LIN {X 0,Y 156.804,Z 513.248,A -85,B 0,C 180,E1 -23850.002,E2 -23850.002} C_VEL
LIN {X 0,Y 156.552,Z 512.223,A -85,B 0,C 180,E1 -23852.575,E2 -23852.575} C_VEL
LIN {X 0,Y 156.139,Z 510.706,A -85,B 0,C 180,E1 -23855.167,E2 -23855.167} C_VEL
LIN {X 0,Y 155.903,Z 507.578,A -85,B 0,C 180,E1 -23859.08,E2 -23859.08} C_VEL
LIN {X 0,Y 156.234,Z 503.359,A -85,B 0,C 180,E1 -23863,E2 -23863} C_VEL
LIN {X 0,Y 157.456,Z 496.901,A -85,B 0,C 180,E1 -23867.537,E2 -23867.537} C_VEL
LIN {X 0,Y 159.345,Z 489.978,A -85,B 0,C 180,E1 -23871.306,E2 -23871.306} C_VEL
LIN {X 0,Y 161.489,Z 483.128,A -85,B 0,C 180,E1 -23874.286,E2 -23874.286} C_VEL
LIN {X 0,Y 162.926,Z 474.015,A -85,B 0,C 180,E1 -23877.629,E2 -23877.629} C_VEL
LIN {X 0,Y 164.364,Z 464.341,A -85,B 0,C 180,E1 -23880.517,E2 -23880.517} C_VEL
LIN {X 0,Y 165.396,Z 453.516,A -85,B 0,C 180,E1 -23883.204,E2 -23883.204} C_VEL
LIN {X 0,Y 165.775,Z 447.367,A -85,B 0,C 180,E1 -23884.528,E2 -23884.528} C_VEL
LIN {X 0,Y 165.255,Z 442.446,A -85,B 0,C 180,E1 -23885.654,E2 -23885.654} C_VEL
LIN {X 0,Y 162.511,Z 434.79,A -85,B 0,C 180,E1 -23887.665,E2 -23887.665} C_VEL
LIN {X 0,Y 159.533,Z 426.921,A -85,B 0,C 180,E1 -23889.587,E2 -23889.587} C_VEL
LIN {X 0,Y 158.608,Z 421.658,A -85,B 0,C 180,E1 -23890.529,E2 -23890.529} C_VEL
LIN {X 0,Y 157.114,Z 411.985,A -85,B 0,C 180,E1 -23892.069,E2 -23892.069} C_VEL
LIN {X 0,Y 154.902,Z 406.011,A -85,B 0,C 180,E1 -23893.256,E2 -23893.256} C_VEL
LIN {X 0,Y 153.361,Z 402.44,A -85,B 0,C 180,E1 -23893.995,E2 -23893.995} C_VEL
LIN {X 0,Y 153.171,Z 401.481,A -85,B 0,C 180,E1 -23894.172,E2 -23894.172} C_VEL
LIN {X 0,Y 152.154,Z 396.368,A -85,B 0,C 180,E1 -23899.71,E2 -23899.71} C_VEL
LIN {X 0,Y 151.356,Z 392.231,A -85,B 0,C 180,E1 -23904.52,E2 -23904.52} C_VEL
LIN {X 0,Y 150.667,Z 388.552,A -85,B 0,C 180,E1 -23909.13,E2 -23909.13} C_VEL
LIN {X 0,Y 150.262,Z 386.768,A -85,B 0,C 180,E1 -23911.735,E2 -23911.735} C_VEL
LIN {X 0,Y 150.274,Z 386.771,A -85,B 0,C 180,E1 -23918.029,E2 -23918.029} C_VEL
LIN {X 0,Y 150.378,Z 386.759,A -85,B 0,C 180,E1 -23920.905,E2 -23920.905} C_VEL
LIN {X 0,Y 150.473,Z 386.744,A -85,B 0,C 180,E1 -23926.496,E2 -23926.496} C_VEL
LIN {X 0,Y 150.695,Z 386.714,A -85,B 0,C 180,E1 -23929.249,E2 -23929.249} C_VEL
LIN {X 0,Y 150.769,Z 386.706,A -85,B 0,C 180,E1 -23931.962,E2 -23931.962} C_VEL
LIN {X 0,Y 151.225,Z 386.636,A -85,B 0,C 180,E1 -23940.001,E2 -23940.001} C_VEL
LIN {X 0,Y 150.767,Z 386.689,A -85,B 0,C 180,E1 -23948.04,E2 -23948.04} C_VEL
LIN {X 0,Y 150.64,Z 386.72,A -85,B 0,C 180,E1 -23951.545,E2 -23951.545} C_VEL
LIN {X 0,Y 150.374,Z 386.739,A -85,B 0,C 180,E1 -23956.286,E2 -23956.286} C_VEL
LIN {X 0,Y 150.357,Z 386.752,A -85,B 0,C 180,E1 -23960.793,E2 -23960.793} C_VEL
LIN {X 0,Y 150.251,Z 386.77,A -85,B 0,C 180,E1 -23967.282,E2 -23967.282} C_VEL
LIN {X 0,Y 150.225,Z 386.771,A -85,B 0,C 180,E1 -23972.634,E2 -23972.634} C_VEL
LIN {X 0,Y 150.217,Z 386.772,A -85,B 0,C 180,E1 -23977.461,E2 -23977.461} C_VEL
LIN {X 0,Y 150.16,Z 386.776,A -85,B 0,C 180,E1 -23981.506,E2 -23981.506} C_VEL
LIN {X 0,Y 150.131,Z 386.78,A -85,B 0,C 180,E1 -23985.395,E2 -23985.395} C_VEL
LIN {X 0,Y 150.156,Z 386.778,A -85,B 0,C 180,E1 -23989.058,E2 -23989.058} C_VEL
LIN {X 0,Y 150.282,Z 386.884,A -85,B 0,C 180,E1 -23994.46,E2 -23994.46} C_VEL
LIN {X 0,Y 151.235,Z 389.587,A -85,B 0,C 180,E1 -23995.172,E2 -23995.172} C_VEL
LIN {X 0,Y 152.671,Z 391.781,A -85,B 0,C 180,E1 -23995.957,E2 -23995.957} C_VEL
LIN {X 0,Y 157.325,Z 400.956,A -85,B 0,C 180,E1 -23998.953,E2 -23998.953} C_VEL
LIN {X 0,Y 161.282,Z 410.794,A -85,B 0,C 180,E1 -24002.092,E2 -24002.092} C_VEL
LIN {X 0,Y 164.08,Z 420.392,A -85,B 0,C 180,E1 -24005.202,E2 -24005.202} C_VEL
LIN {X 0,Y 165.343,Z 425.976,A -85,B 0,C 180,E1 -24007.113,E2 -24007.113} C_VEL
LIN {X 0,Y 162.841,Z 435.568,A -85,B 0,C 180,E1 -24009.8,E2 -24009.8} C_VEL
LIN {X 0,Y 160.103,Z 444.185,A -85,B 0,C 180,E1 -24012.762,E2 -24012.762} C_VEL
LIN {X 0,Y 157.588,Z 451.322,A -85,B 0,C 180,E1 -24015.799,E2 -24015.799} C_VEL
LIN {X 0,Y 155.089,Z 458.345,A -85,B 0,C 180,E1 -24019.555,E2 -24019.555} C_VEL
LIN {X 0,Y 153.157,Z 463.944,A -85,B 0,C 180,E1 -24023.411,E2 -24023.411} C_VEL
LIN {X 0,Y 151.613,Z 468.389,A -85,B 0,C 180,E1 -24027.341,E2 -24027.341} C_VEL
LIN {X 0,Y 150.875,Z 470.747,A -85,B 0,C 180,E1 -24029.998,E2 -24029.998} C_VEL
LIN {X 0,Y 150.369,Z 472.687,A -85,B 0,C 180,E1 -24032.677,E2 -24032.677} C_VEL
LIN {X 0,Y 150.284,Z 474.186,A -85,B 0,C 180,E1 -24035.365,E2 -24035.365} C_VEL
LIN {X 0,Y 150.347,Z 475.258,A -85,B 0,C 180,E1 -24038.06,E2 -24038.06} C_VEL
LIN {X 0,Y 151.03,Z 476.287,A -85,B 0,C 180,E1 -24043.452,E2 -24043.452} C_VEL
LIN {X 0,Y 151.721,Z 476.222,A -85,B 0,C 180,E1 -24046.135,E2 -24046.135} C_VEL
LIN {X 0,Y 153.88,Z 474.85,A -85,B 0,C 180,E1 -24051.429,E2 -24051.429} C_VEL
LIN {X 0,Y 155.422,Z 473.57,A -85,B 0,C 180,E1 -24054.012,E2 -24054.012} C_VEL
LIN {X 0,Y 158.105,Z 470.825,A -85,B 0,C 180,E1 -24057.821,E2 -24057.821} C_VEL
LIN {X 0,Y 161.348,Z 467.038,A -85,B 0,C 180,E1 -24061.511,E2 -24061.511} C_VEL
LIN {X 0,Y 165.108,Z 462.098,A -85,B 0,C 180,E1 -24065.072,E2 -24065.072} C_VEL
LIN {X 0,Y 169.45,Z 455.8,A -85,B 0,C 180,E1 -24068.47,E2 -24068.47} C_VEL
LIN {X 0,Y 174.228,Z 447.87,A -85,B 0,C 180,E1 -24071.724,E2 -24071.724} C_VEL
LIN {X 0,Y 175.852,Z 444.813,A -85,B 0,C 180,E1 -24072.795,E2 -24072.795} C_VEL
LIN {X 0,Y 175.242,Z 438.143,A -85,B 0,C 180,E1 -24076.208,E2 -24076.208} C_VEL
LIN {X 0,Y 173.539,Z 430.026,A -85,B 0,C 180,E1 -24080.303,E2 -24080.303} C_VEL
LIN {X 0,Y 171.262,Z 422.341,A -85,B 0,C 180,E1 -24084.212,E2 -24084.212} C_VEL
LIN {X 0,Y 168.083,Z 414.609,A -85,B 0,C 180,E1 -24088.488,E2 -24088.488} C_VEL
LIN {X 0,Y 164.176,Z 406.916,A -85,B 0,C 180,E1 -24093.289,E2 -24093.289} C_VEL
LIN {X 0,Y 161.151,Z 402.126,A -85,B 0,C 180,E1 -24096.889,E2 -24096.889} C_VEL
LIN {X 0,Y 159.253,Z 399.15,A -85,B 0,C 180,E1 -24099.325,E2 -24099.325} C_VEL
LIN {X 0,Y 158.101,Z 397.442,A -85,B 0,C 180,E1 -24100.862,E2 -24100.862} C_VEL
LIN {X 0,Y 156.068,Z 395.021,A -85,B 0,C 180,E1 -24103.653,E2 -24103.653} C_VEL
LIN {X 0,Y 155.062,Z 392.527,A -85,B 0,C 180,E1 -24105.564,E2 -24105.564} C_VEL
LIN {X 0,Y 152.252,Z 390.308,A -85,B 0,C 180,E1 -24110.367,E2 -24110.367} C_VEL
LIN {X 0,Y 150.758,Z 387.15,A -85,B 0,C 180,E1 -24114.817,E2 -24114.817} C_VEL
LIN {X 0,Y 150.713,Z 386.693,A -85,B 0,C 180,E1 -24115.319,E2 -24115.319} C_VEL
LIN {X 0,Y 151.218,Z 386.63,A -85,B 0,C 180,E1 -24119.999,E2 -24119.999} C_VEL
LIN {X 0,Y 150.955,Z 386.816,A -85,B 0,C 180,E1 -24122.668,E2 -24122.668} C_VEL
LIN {X 0,Y 151.141,Z 388.563,A -85,B 0,C 180,E1 -24128.018,E2 -24128.018} C_VEL
LIN {X 0,Y 151.34,Z 389.576,A -85,B 0,C 180,E1 -24130.705,E2 -24130.705} C_VEL
LIN {X 0,Y 151.465,Z 391.249,A -85,B 0,C 180,E1 -24134.099,E2 -24134.099} C_VEL
LIN {X 0,Y 154.139,Z 397.245,A -85,B 0,C 180,E1 -24139.649,E2 -24139.649} C_VEL
LIN {X 0,Y 156.992,Z 401.179,A -85,B 0,C 180,E1 -24143.54,E2 -24143.54} C_VEL
LIN {X 0,Y 158.698,Z 405.379,A -85,B 0,C 180,E1 -24145.932,E2 -24145.932} C_VEL
LIN {X 0,Y 161.296,Z 409.223,A -85,B 0,C 180,E1 -24148.69,E2 -24148.69} C_VEL
LIN {X 0,Y 163.364,Z 414.032,A -85,B 0,C 180,E1 -24151.08,E2 -24151.08} C_VEL
LIN {X 0,Y 164.608,Z 416.098,A -85,B 0,C 180,E1 -24152.255,E2 -24152.255} C_VEL
LIN {X 0,Y 165.981,Z 419.751,A -85,B 0,C 180,E1 -24153.832,E2 -24153.832} C_VEL
LIN {X 0,Y 167.386,Z 422.972,A -85,B 0,C 180,E1 -24155.262,E2 -24155.262} C_VEL
LIN {X 0,Y 169.635,Z 429.16,A -85,B 0,C 180,E1 -24157.744,E2 -24157.744} C_VEL
LIN {X 0,Y 172.193,Z 437.216,A -85,B 0,C 180,E1 -24160.77,E2 -24160.77} C_VEL
LIN {X 0,Y 172.884,Z 439.902,A -85,B 0,C 180,E1 -24161.71,E2 -24161.71} C_VEL
LIN {X 0,Y 172.455,Z 450.46,A -85,B 0,C 180,E1 -24164.471,E2 -24164.471} C_VEL
LIN {X 0,Y 171.024,Z 461.95,A -85,B 0,C 180,E1 -24167.704,E2 -24167.704} C_VEL
LIN {X 0,Y 169.027,Z 471.309,A -85,B 0,C 180,E1 -24170.65,E2 -24170.65} C_VEL
LIN {X 0,Y 166.508,Z 479.96,A -85,B 0,C 180,E1 -24173.78,E2 -24173.78} C_VEL
LIN {X 0,Y 163.75,Z 487.195,A -85,B 0,C 180,E1 -24176.826,E2 -24176.826} C_VEL
LIN {X 0,Y 160.277,Z 493.196,A -85,B 0,C 180,E1 -24179.72,E2 -24179.72} C_VEL
LIN {X 0,Y 156.417,Z 499.094,A -85,B 0,C 180,E1 -24183.303,E2 -24183.303} C_VEL
LIN {X 0,Y 153.318,Z 503.813,A -85,B 0,C 180,E1 -24187.07,E2 -24187.07} C_VEL
LIN {X 0,Y 151.006,Z 507.478,A -85,B 0,C 180,E1 -24190.989,E2 -24190.989} C_VEL
LIN {X 0,Y 149.135,Z 510.845,A -85,B 0,C 180,E1 -24196.374,E2 -24196.374} C_VEL
LIN {X 0,Y 148.732,Z 512.676,A -85,B 0,C 180,E1 -24201.852,E2 -24201.852} C_VEL
LIN {X 0,Y 148.981,Z 512.974,A -85,B 0,C 180,E1 -24204.588,E2 -24204.588} C_VEL
LIN {X 0,Y 149.486,Z 512.875,A -85,B 0,C 180,E1 -24207.307,E2 -24207.307} C_VEL
LIN {X 0,Y 149.755,Z 512.326,A -85,B 0,C 180,E1 -24210.002,E2 -24210.002} C_VEL
LIN {X 0,Y 149.455,Z 511.273,A -85,B 0,C 180,E1 -24212.697,E2 -24212.697} C_VEL
LIN {X 0,Y 148.909,Z 508.114,A -85,B 0,C 180,E1 -24217.64,E2 -24217.64} C_VEL
LIN {X 0,Y 149.055,Z 503.801,A -85,B 0,C 180,E1 -24222.252,E2 -24222.252} C_VEL
LIN {X 0,Y 149.915,Z 498.753,A -85,B 0,C 180,E1 -24226.339,E2 -24226.339} C_VEL
LIN {X 0,Y 151.489,Z 492.41,A -85,B 0,C 180,E1 -24230.364,E2 -24230.364} C_VEL
LIN {X 0,Y 154.137,Z 484.605,A -85,B 0,C 180,E1 -24234.23,E2 -24234.23} C_VEL
LIN {X 0,Y 155.227,Z 479.875,A -85,B 0,C 180,E1 -24236.198,E2 -24236.198} C_VEL
LIN {X 0,Y 156.894,Z 469.535,A -85,B 0,C 180,E1 -24239.892,E2 -24239.892} C_VEL
LIN {X 0,Y 158.385,Z 459.298,A -85,B 0,C 180,E1 -24242.853,E2 -24242.853} C_VEL
LIN {X 0,Y 159.327,Z 448.053,A -85,B 0,C 180,E1 -24245.558,E2 -24245.558} C_VEL
LIN {X 0,Y 159.587,Z 437.505,A -85,B 0,C 180,E1 -24247.724,E2 -24247.724} C_VEL
LIN {X 0,Y 158.895,Z 424.497,A -85,B 0,C 180,E1 -24250.053,E2 -24250.053} C_VEL
LIN {X 0,Y 158.608,Z 421.658,A -85,B 0,C 180,E1 -24250.529,E2 -24250.529} C_VEL
LIN {X 0,Y 157.656,Z 418.369,A -85,B 0,C 180,E1 -24251.197,E2 -24251.197} C_VEL
LIN {X 0,Y 155.771,Z 415.711,A -85,B 0,C 180,E1 -24252.036,E2 -24252.036} C_VEL
LIN {X 0,Y 150.382,Z 410.253,A -85,B 0,C 180,E1 -24254.212,E2 -24254.212} C_VEL
LIN {X 0,Y 148.643,Z 407.257,A -85,B 0,C 180,E1 -24255.055,E2 -24255.055} C_VEL
LIN {X 0,Y 147.84,Z 405.365,A -85,B 0,C 180,E1 -24255.501,E2 -24255.501} C_VEL
LIN {X 0,Y 146.067,Z 401.9,A -85,B 0,C 180,E1 -24256.411,E2 -24256.411} C_VEL
LIN {X 0,Y 145.648,Z 400.322,A -85,B 0,C 180,E1 -24256.731,E2 -24256.731} C_VEL
LIN {X 0,Y 144.703,Z 395.265,A -85,B 0,C 180,E1 -24262.62,E2 -24262.62} C_VEL
LIN {X 0,Y 143.976,Z 391.441,A -85,B 0,C 180,E1 -24267.524,E2 -24267.524} C_VEL
LIN {X 0,Y 143.217,Z 387.647,A -85,B 0,C 180,E1 -24272.877,E2 -24272.877} C_VEL
LIN {X 0,Y 143.318,Z 387.638,A -85,B 0,C 180,E1 -24279.925,E2 -24279.925} C_VEL
LIN {X 0,Y 143.39,Z 387.627,A -85,B 0,C 180,E1 -24285.815,E2 -24285.815} C_VEL
LIN {X 0,Y 143.609,Z 387.599,A -85,B 0,C 180,E1 -24288.712,E2 -24288.712} C_VEL
LIN {X 0,Y 143.691,Z 387.587,A -85,B 0,C 180,E1 -24291.563,E2 -24291.563} C_VEL
LIN {X 0,Y 144.183,Z 387.512,A -85,B 0,C 180,E1 -24300.001,E2 -24300.001} C_VEL
LIN {X 0,Y 143.689,Z 387.572,A -85,B 0,C 180,E1 -24308.438,E2 -24308.438} C_VEL
LIN {X 0,Y 143.578,Z 387.599,A -85,B 0,C 180,E1 -24311.758,E2 -24311.758} C_VEL
LIN {X 0,Y 143.312,Z 387.625,A -85,B 0,C 180,E1 -24317.113,E2 -24317.113} C_VEL
LIN {X 0,Y 143.283,Z 387.628,A -85,B 0,C 180,E1 -24321.255,E2 -24321.255} C_VEL
LIN {X 0,Y 143.197,Z 387.645,A -85,B 0,C 180,E1 -24327.937,E2 -24327.937} C_VEL
LIN {X 0,Y 143.175,Z 387.651,A -85,B 0,C 180,E1 -24333.435,E2 -24333.435} C_VEL
LIN {X 0,Y 143.081,Z 387.66,A -85,B 0,C 180,E1 -24339.685,E2 -24339.685} C_VEL
LIN {X 0,Y 143.062,Z 387.662,A -85,B 0,C 180,E1 -24343.454,E2 -24343.454} C_VEL
LIN {X 0,Y 143.071,Z 387.658,A -85,B 0,C 180,E1 -24347.464,E2 -24347.464} C_VEL
LIN {X 0,Y 143.097,Z 387.656,A -85,B 0,C 180,E1 -24351.945,E2 -24351.945} C_VEL
LIN {X 0,Y 144.15,Z 390.466,A -85,B 0,C 180,E1 -24352.795,E2 -24352.795} C_VEL
LIN {X 0,Y 145.692,Z 392.601,A -85,B 0,C 180,E1 -24353.701,E2 -24353.701} C_VEL
LIN {X 0,Y 150.599,Z 402.137,A -85,B 0,C 180,E1 -24357.142,E2 -24357.142} C_VEL
LIN {X 0,Y 154.538,Z 411.723,A -85,B 0,C 180,E1 -24360.481,E2 -24360.481} C_VEL
LIN {X 0,Y 157.134,Z 420.241,A -85,B 0,C 180,E1 -24363.449,E2 -24363.449} C_VEL
LIN {X 0,Y 158.795,Z 427.615,A -85,B 0,C 180,E1 -24366.121,E2 -24366.121} C_VEL
LIN {X 0,Y 158.105,Z 431.034,A -85,B 0,C 180,E1 -24367.109,E2 -24367.109} C_VEL
LIN {X 0,Y 155.103,Z 440.619,A -85,B 0,C 180,E1 -24370.131,E2 -24370.131} C_VEL
LIN {X 0,Y 152.287,Z 448.512,A -85,B 0,C 180,E1 -24373.234,E2 -24373.234} C_VEL
LIN {X 0,Y 149.363,Z 456.267,A -85,B 0,C 180,E1 -24377.083,E2 -24377.083} C_VEL
LIN {X 0,Y 147.406,Z 461.521,A -85,B 0,C 180,E1 -24380.392,E2 -24380.392} C_VEL
LIN {X 0,Y 145.544,Z 466.668,A -85,B 0,C 180,E1 -24384.456,E2 -24384.456} C_VEL
LIN {X 0,Y 144.157,Z 470.694,A -85,B 0,C 180,E1 -24388.601,E2 -24388.601} C_VEL
LIN {X 0,Y 143.307,Z 473.698,A -85,B 0,C 180,E1 -24392.809,E2 -24392.809} C_VEL
LIN {X 0,Y 143.248,Z 475.147,A -85,B 0,C 180,E1 -24395.629,E2 -24395.629} C_VEL
LIN {X 0,Y 143.334,Z 476.194,A -85,B 0,C 180,E1 -24398.457,E2 -24398.457} C_VEL
LIN {X 0,Y 143.738,Z 477.012,A -85,B 0,C 180,E1 -24402.065,E2 -24402.065} C_VEL
LIN {X 0,Y 144.895,Z 477.065,A -85,B 0,C 180,E1 -24406.917,E2 -24406.917} C_VEL
LIN {X 0,Y 147.256,Z 475.645,A -85,B 0,C 180,E1 -24412.444,E2 -24412.444} C_VEL
LIN {X 0,Y 148.937,Z 474.336,A -85,B 0,C 180,E1 -24415.129,E2 -24415.129} C_VEL
LIN {X 0,Y 151.811,Z 471.544,A -85,B 0,C 180,E1 -24419.082,E2 -24419.082} C_VEL
LIN {X 0,Y 155.297,Z 467.7,A -85,B 0,C 180,E1 -24422.89,E2 -24422.89} C_VEL
LIN {X 0,Y 159.315,Z 462.688,A -85,B 0,C 180,E1 -24426.549,E2 -24426.549} C_VEL
LIN {X 0,Y 163.9,Z 456.301,A -85,B 0,C 180,E1 -24430.028,E2 -24430.028} C_VEL
LIN {X 0,Y 168.941,Z 448.293,A -85,B 0,C 180,E1 -24433.344,E2 -24433.344} C_VEL
LIN {X 0,Y 169.553,Z 447.247,A -85,B 0,C 180,E1 -24433.729,E2 -24433.729} C_VEL
LIN {X 0,Y 169.328,Z 441.657,A -85,B 0,C 180,E1 -24436.776,E2 -24436.776} C_VEL
LIN {X 0,Y 167.965,Z 433.738,A -85,B 0,C 180,E1 -24441.124,E2 -24441.124} C_VEL
LIN {X 0,Y 166.301,Z 427.219,A -85,B 0,C 180,E1 -24444.714,E2 -24444.714} C_VEL
LIN {X 0,Y 163.721,Z 420.023,A -85,B 0,C 180,E1 -24448.994,E2 -24448.994} C_VEL
LIN {X 0,Y 160.324,Z 412.549,A -85,B 0,C 180,E1 -24454,E2 -24454} C_VEL
LIN {X 0,Y 158.581,Z 409.271,A -85,B 0,C 180,E1 -24456.492,E2 -24456.492} C_VEL
LIN {X 0,Y 156.76,Z 406.615,A -85,B 0,C 180,E1 -24458.981,E2 -24458.981} C_VEL
LIN {X 0,Y 156.056,Z 404.955,A -85,B 0,C 180,E1 -24460.259,E2 -24460.259} C_VEL
LIN {X 0,Y 153.616,Z 401.624,A -85,B 0,C 180,E1 -24464.067,E2 -24464.067} C_VEL
LIN {X 0,Y 152.809,Z 399.243,A -85,B 0,C 180,E1 -24466.027,E2 -24466.027} C_VEL
LIN {X 0,Y 150.099,Z 396.609,A -85,B 0,C 180,E1 -24471.586,E2 -24471.586} C_VEL
LIN {X 0,Y 149.103,Z 393.584,A -85,B 0,C 180,E1 -24475.945,E2 -24475.945} C_VEL
LIN {X 0,Y 148.204,Z 393.163,A -85,B 0,C 180,E1 -24481.358,E2 -24481.358} C_VEL
LIN {X 0,Y 148.406,Z 395.088,A -85,B 0,C 180,E1 -24487.825,E2 -24487.825} C_VEL
LIN {X 0,Y 149.836,Z 397.865,A -85,B 0,C 180,E1 -24493.261,E2 -24493.261} C_VEL
LIN {X 0,Y 152.82,Z 404.973,A -85,B 0,C 180,E1 -24500.176,E2 -24500.176} C_VEL
LIN {X 0,Y 154.443,Z 407.392,A -85,B 0,C 180,E1 -24502.578,E2 -24502.578} C_VEL
LIN {X 0,Y 155.993,Z 411.564,A -85,B 0,C 180,E1 -24505.163,E2 -24505.163} C_VEL
LIN {X 0,Y 158.129,Z 415.28,A -85,B 0,C 180,E1 -24507.818,E2 -24507.818} C_VEL
LIN {X 0,Y 160.188,Z 420.206,A -85,B 0,C 180,E1 -24510.515,E2 -24510.515} C_VEL
LIN {X 0,Y 161.044,Z 422.241,A -85,B 0,C 180,E1 -24511.579,E2 -24511.579} C_VEL
LIN {X 0,Y 163.538,Z 429.156,A -85,B 0,C 180,E1 -24514.811,E2 -24514.811} C_VEL
LIN {X 0,Y 166.171,Z 437.681,A -85,B 0,C 180,E1 -24518.411,E2 -24518.411} C_VEL
LIN {X 0,Y 167.504,Z 443.254,A -85,B 0,C 180,E1 -24520.568,E2 -24520.568} C_VEL
LIN {X 0,Y 166.782,Z 452.813,A -85,B 0,C 180,E1 -24523.283,E2 -24523.283} C_VEL
LIN {X 0,Y 165.143,Z 462.953,A -85,B 0,C 180,E1 -24526.341,E2 -24526.341} C_VEL
LIN {X 0,Y 162.728,Z 472.698,A -85,B 0,C 180,E1 -24529.624,E2 -24529.624} C_VEL
LIN {X 0,Y 160.014,Z 480.978,A -85,B 0,C 180,E1 -24532.851,E2 -24532.851} C_VEL
LIN {X 0,Y 157.08,Z 487.892,A -85,B 0,C 180,E1 -24535.997,E2 -24535.997} C_VEL
LIN {X 0,Y 152.738,Z 494.658,A -85,B 0,C 180,E1 -24539.595,E2 -24539.595} C_VEL
LIN {X 0,Y 148.906,Z 500.101,A -85,B 0,C 180,E1 -24543.364,E2 -24543.364} C_VEL
LIN {X 0,Y 145.839,Z 504.401,A -85,B 0,C 180,E1 -24547.326,E2 -24547.326} C_VEL
LIN {X 0,Y 144.269,Z 506.714,A -85,B 0,C 180,E1 -24550.064,E2 -24550.064} C_VEL
LIN {X 0,Y 142.177,Z 510.029,A -85,B 0,C 180,E1 -24555.693,E2 -24555.693} C_VEL
LIN {X 0,Y 141.666,Z 511.811,A -85,B 0,C 180,E1 -24561.443,E2 -24561.443} C_VEL
LIN {X 0,Y 142.393,Z 511.966,A -85,B 0,C 180,E1 -24567.173,E2 -24567.173} C_VEL
LIN {X 0,Y 142.704,Z 511.404,A -85,B 0,C 180,E1 -24570.002,E2 -24570.002} C_VEL
LIN {X 0,Y 142.359,Z 510.317,A -85,B 0,C 180,E1 -24572.832,E2 -24572.832} C_VEL
LIN {X 0,Y 141.832,Z 507.361,A -85,B 0,C 180,E1 -24577.681,E2 -24577.681} C_VEL
LIN {X 0,Y 142.056,Z 502.734,A -85,B 0,C 180,E1 -24582.866,E2 -24582.866} C_VEL
LIN {X 0,Y 143.029,Z 497.633,A -85,B 0,C 180,E1 -24587.149,E2 -24587.149} C_VEL
LIN {X 0,Y 144.806,Z 491.241,A -85,B 0,C 180,E1 -24591.349,E2 -24591.349} C_VEL
LIN {X 0,Y 147.617,Z 483.339,A -85,B 0,C 180,E1 -24595.374,E2 -24595.374} C_VEL
LIN {X 0,Y 149.198,Z 474.986,A -85,B 0,C 180,E1 -24598.873,E2 -24598.873} C_VEL
LIN {X 0,Y 151.014,Z 465.092,A -85,B 0,C 180,E1 -24602.245,E2 -24602.245} C_VEL
LIN {X 0,Y 152.358,Z 454.626,A -85,B 0,C 180,E1 -24605.214,E2 -24605.214} C_VEL
LIN {X 0,Y 153.249,Z 443.066,A -85,B 0,C 180,E1 -24607.956,E2 -24607.956} C_VEL
LIN {X 0,Y 153.206,Z 431.117,A -85,B 0,C 180,E1 -24610.39,E2 -24610.39} C_VEL
LIN {X 0,Y 152.052,Z 417.733,A -85,B 0,C 180,E1 -24612.798,E2 -24612.798} C_VEL
LIN {X 0,Y 151.084,Z 413.443,A -85,B 0,C 180,E1 -24613.621,E2 -24613.621} C_VEL
LIN {X 0,Y 149.392,Z 409.074,A -85,B 0,C 180,E1 -24614.64,E2 -24614.64} C_VEL
LIN {X 0,Y 148.643,Z 407.257,A -85,B 0,C 180,E1 -24615.055,E2 -24615.055} C_VEL
LIN {X 0,Y 146.916,Z 404.352,A -85,B 0,C 180,E1 -24615.915,E2 -24615.915} C_VEL
LIN {X 0,Y 143.683,Z 401.629,A -85,B 0,C 180,E1 -24617.283,E2 -24617.283} C_VEL
LIN {X 0,Y 139.622,Z 399.318,A -85,B 0,C 180,E1 -24619.339,E2 -24619.339} C_VEL
LIN {X 0,Y 138.129,Z 398.107,A -85,B 0,C 180,E1 -24620.82,E2 -24620.82} C_VEL
LIN {X 0,Y 137.944,Z 397.693,A -85,B 0,C 180,E1 -24621.351,E2 -24621.351} C_VEL
LIN {X 0,Y 137.081,Z 393.137,A -85,B 0,C 180,E1 -24627.431,E2 -24627.431} C_VEL
LIN {X 0,Y 136.392,Z 389.758,A -85,B 0,C 180,E1 -24632.371,E2 -24632.371} C_VEL
LIN {X 0,Y 136.1,Z 388.535,A -85,B 0,C 180,E1 -24634.376,E2 -24634.376} C_VEL
LIN {X 0,Y 136.25,Z 388.519,A -85,B 0,C 180,E1 -24638.835,E2 -24638.835} C_VEL
LIN {X 0,Y 136.295,Z 388.51,A -85,B 0,C 180,E1 -24645.06,E2 -24645.06} C_VEL
LIN {X 0,Y 136.507,Z 388.482,A -85,B 0,C 180,E1 -24648.116,E2 -24648.116} C_VEL
LIN {X 0,Y 136.614,Z 388.468,A -85,B 0,C 180,E1 -24651.123,E2 -24651.123} C_VEL
LIN {X 0,Y 137.141,Z 388.389,A -85,B 0,C 180,E1 -24660.001,E2 -24660.001} C_VEL
LIN {X 0,Y 136.613,Z 388.457,A -85,B 0,C 180,E1 -24668.879,E2 -24668.879} C_VEL
LIN {X 0,Y 136.498,Z 388.479,A -85,B 0,C 180,E1 -24671.956,E2 -24671.956} C_VEL
LIN {X 0,Y 136.251,Z 388.509,A -85,B 0,C 180,E1 -24678.029,E2 -24678.029} C_VEL
LIN {X 0,Y 136.205,Z 388.505,A -85,B 0,C 180,E1 -24681.749,E2 -24681.749} C_VEL
LIN {X 0,Y 136.107,Z 388.523,A -85,B 0,C 180,E1 -24688.616,E2 -24688.616} C_VEL
LIN {X 0,Y 136.085,Z 388.532,A -85,B 0,C 180,E1 -24694.618,E2 -24694.618} C_VEL
LIN {X 0,Y 136.057,Z 388.533,A -85,B 0,C 180,E1 -24699.208,E2 -24699.208} C_VEL
LIN {X 0,Y 136.004,Z 388.54,A -85,B 0,C 180,E1 -24703.657,E2 -24703.657} C_VEL
LIN {X 0,Y 136.016,Z 388.723,A -85,B 0,C 180,E1 -24709.156,E2 -24709.156} C_VEL
LIN {X 0,Y 137.055,Z 391.43,A -85,B 0,C 180,E1 -24710.076,E2 -24710.076} C_VEL
LIN {X 0,Y 138.599,Z 393.145,A -85,B 0,C 180,E1 -24711.029,E2 -24711.029} C_VEL
LIN {X 0,Y 139.758,Z 395.667,A -85,B 0,C 180,E1 -24711.974,E2 -24711.974} C_VEL
LIN {X 0,Y 142.844,Z 401.142,A -85,B 0,C 180,E1 -24714.272,E2 -24714.272} C_VEL
LIN {X 0,Y 146.71,Z 409.736,A -85,B 0,C 180,E1 -24717.602,E2 -24717.602} C_VEL
LIN {X 0,Y 149.787,Z 418.545,A -85,B 0,C 180,E1 -24720.932,E2 -24720.932} C_VEL
LIN {X 0,Y 151.862,Z 427.073,A -85,B 0,C 180,E1 -24724.18,E2 -24724.18} C_VEL
LIN {X 0,Y 152.349,Z 430.442,A -85,B 0,C 180,E1 -24725.467,E2 -24725.467} C_VEL
LIN {X 0,Y 149.138,Z 440.275,A -85,B 0,C 180,E1 -24728.577,E2 -24728.577} C_VEL
LIN {X 0,Y 145.562,Z 449.836,A -85,B 0,C 180,E1 -24732.434,E2 -24732.434} C_VEL
LIN {X 0,Y 142.509,Z 457.479,A -85,B 0,C 180,E1 -24736.45,E2 -24736.45} C_VEL
LIN {X 0,Y 139.771,Z 464.494,A -85,B 0,C 180,E1 -24741.322,E2 -24741.322} C_VEL
LIN {X 0,Y 138.004,Z 469.192,A -85,B 0,C 180,E1 -24745.617,E2 -24745.617} C_VEL
LIN {X 0,Y 136.711,Z 472.824,A -85,B 0,C 180,E1 -24749.998,E2 -24749.998} C_VEL
LIN {X 0,Y 136.247,Z 474.704,A -85,B 0,C 180,E1 -24752.955,E2 -24752.955} C_VEL
LIN {X 0,Y 136.215,Z 476.106,A -85,B 0,C 180,E1 -24755.921,E2 -24755.921} C_VEL
LIN {X 0,Y 136.634,Z 477.79,A -85,B 0,C 180,E1 -24761.871,E2 -24761.871} C_VEL
LIN {X 0,Y 137.219,Z 478.064,A -85,B 0,C 180,E1 -24764.836,E2 -24764.836} C_VEL
LIN {X 0,Y 139.243,Z 477.367,A -85,B 0,C 180,E1 -24770.688,E2 -24770.688} C_VEL
LIN {X 0,Y 140.684,Z 476.44,A -85,B 0,C 180,E1 -24773.554,E2 -24773.554} C_VEL
LIN {X 0,Y 144.191,Z 473.603,A -85,B 0,C 180,E1 -24778.675,E2 -24778.675} C_VEL
LIN {X 0,Y 148.035,Z 469.751,A -85,B 0,C 180,E1 -24783.088,E2 -24783.088} C_VEL
LIN {X 0,Y 152.119,Z 465.081,A -85,B 0,C 180,E1 -24786.911,E2 -24786.911} C_VEL
LIN {X 0,Y 156.842,Z 459.087,A -85,B 0,C 180,E1 -24790.543,E2 -24790.543} C_VEL
LIN {X 0,Y 161.996,Z 451.645,A -85,B 0,C 180,E1 -24793.956,E2 -24793.956} C_VEL
LIN {X 0,Y 163.463,Z 449.155,A -85,B 0,C 180,E1 -24794.931,E2 -24794.931} C_VEL
LIN {X 0,Y 163.239,Z 443.902,A -85,B 0,C 180,E1 -24798.106,E2 -24798.106} C_VEL
LIN {X 0,Y 162.433,Z 437.767,A -85,B 0,C 180,E1 -24801.757,E2 -24801.757} C_VEL
LIN {X 0,Y 161.106,Z 431.601,A -85,B 0,C 180,E1 -24805.45,E2 -24805.45} C_VEL
LIN {X 0,Y 159.321,Z 425.709,A -85,B 0,C 180,E1 -24809.231,E2 -24809.231} C_VEL
LIN {X 0,Y 156.373,Z 418.222,A -85,B 0,C 180,E1 -24814.581,E2 -24814.581} C_VEL
LIN {X 0,Y 154.788,Z 414.926,A -85,B 0,C 180,E1 -24817.297,E2 -24817.297} C_VEL
LIN {X 0,Y 152.639,Z 410.761,A -85,B 0,C 180,E1 -24821.197,E2 -24821.197} C_VEL
LIN {X 0,Y 150.824,Z 408.059,A -85,B 0,C 180,E1 -24824.538,E2 -24824.538} C_VEL
LIN {X 0,Y 150.202,Z 405.981,A -85,B 0,C 180,E1 -24826.469,E2 -24826.469} C_VEL
LIN {X 0,Y 148.003,Z 403.38,A -85,B 0,C 180,E1 -24831.809,E2 -24831.809} C_VEL
LIN {X 0,Y 147.202,Z 400.407,A -85,B 0,C 180,E1 -24836.578,E2 -24836.578} C_VEL
LIN {X 0,Y 146.623,Z 400.059,A -85,B 0,C 180,E1 -24841.373,E2 -24841.373} C_VEL
LIN {X 0,Y 147.142,Z 402.834,A -85,B 0,C 180,E1 -24849.623,E2 -24849.623} C_VEL
LIN {X 0,Y 147.918,Z 404.617,A -85,B 0,C 180,E1 -24852.694,E2 -24852.694} C_VEL
LIN {X 0,Y 150.178,Z 411.023,A -85,B 0,C 180,E1 -24859.122,E2 -24859.122} C_VEL
LIN {X 0,Y 151.639,Z 413.697,A -85,B 0,C 180,E1 -24861.763,E2 -24861.763} C_VEL
LIN {X 0,Y 153.003,Z 417.653,A -85,B 0,C 180,E1 -24864.418,E2 -24864.418} C_VEL
LIN {X 0,Y 154.743,Z 421.203,A -85,B 0,C 180,E1 -24867.011,E2 -24867.011} C_VEL
LIN {X 0,Y 156.887,Z 426.748,A -85,B 0,C 180,E1 -24870.262,E2 -24870.262} C_VEL
LIN {X 0,Y 159.734,Z 436.145,A -85,B 0,C 180,E1 -24874.888,E2 -24874.888} C_VEL
LIN {X 0,Y 161.748,Z 444.501,A -85,B 0,C 180,E1 -24878.549,E2 -24878.549} C_VEL
LIN {X 0,Y 162.146,Z 446.757,A -85,B 0,C 180,E1 -24879.487,E2 -24879.487} C_VEL
LIN {X 0,Y 160.831,Z 456.624,A -85,B 0,C 180,E1 -24882.492,E2 -24882.492} C_VEL
LIN {X 0,Y 158.929,Z 465.671,A -85,B 0,C 180,E1 -24885.472,E2 -24885.472} C_VEL
LIN {X 0,Y 155.915,Z 475.7,A -85,B 0,C 180,E1 -24889.189,E2 -24889.189} C_VEL
LIN {X 0,Y 152.963,Z 483.341,A -85,B 0,C 180,E1 -24892.505,E2 -24892.505} C_VEL
LIN {X 0,Y 149.698,Z 489.716,A -85,B 0,C 180,E1 -24895.713,E2 -24895.713} C_VEL
LIN {X 0,Y 145.162,Z 495.939,A -85,B 0,C 180,E1 -24899.448,E2 -24899.448} C_VEL
LIN {X 0,Y 141.161,Z 501.193,A -85,B 0,C 180,E1 -24903.658,E2 -24903.658} C_VEL
LIN {X 0,Y 138.348,Z 504.844,A -85,B 0,C 180,E1 -24907.607,E2 -24907.607} C_VEL
LIN {X 0,Y 136.177,Z 507.769,A -85,B 0,C 180,E1 -24911.964,E2 -24911.964} C_VEL
LIN {X 0,Y 134.74,Z 510.283,A -85,B 0,C 180,E1 -24917.96,E2 -24917.96} C_VEL
LIN {X 0,Y 134.807,Z 511.19,A -85,B 0,C 180,E1 -24924.017,E2 -24924.017} C_VEL
LIN {X 0,Y 135.302,Z 511.057,A -85,B 0,C 180,E1 -24927.025,E2 -24927.025} C_VEL
LIN {X 0,Y 135.651,Z 510.48,A -85,B 0,C 180,E1 -24930.002,E2 -24930.002} C_VEL
LIN {X 0,Y 135.265,Z 509.351,A -85,B 0,C 180,E1 -24932.98,E2 -24932.98} C_VEL
LIN {X 0,Y 134.77,Z 506.572,A -85,B 0,C 180,E1 -24937.775,E2 -24937.775} C_VEL
LIN {X 0,Y 135.086,Z 501.664,A -85,B 0,C 180,E1 -24943.542,E2 -24943.542} C_VEL
LIN {X 0,Y 136.46,Z 495.548,A -85,B 0,C 180,E1 -24948.779,E2 -24948.779} C_VEL
LIN {X 0,Y 138.65,Z 488.842,A -85,B 0,C 180,E1 -24953.134,E2 -24953.134} C_VEL
LIN {X 0,Y 141.071,Z 482.047,A -85,B 0,C 180,E1 -24956.642,E2 -24956.642} C_VEL
LIN {X 0,Y 142.719,Z 473.584,A -85,B 0,C 180,E1 -24960.317,E2 -24960.317} C_VEL
LIN {X 0,Y 144.556,Z 464.38,A -85,B 0,C 180,E1 -24963.578,E2 -24963.578} C_VEL
LIN {X 0,Y 146.02,Z 454.348,A -85,B 0,C 180,E1 -24966.559,E2 -24966.559} C_VEL
LIN {X 0,Y 147.036,Z 442.36,A -85,B 0,C 180,E1 -24969.567,E2 -24969.567} C_VEL
LIN {X 0,Y 147.075,Z 430.057,A -85,B 0,C 180,E1 -24972.21,E2 -24972.21} C_VEL
LIN {X 0,Y 146.067,Z 418.013,A -85,B 0,C 180,E1 -24974.548,E2 -24974.548} C_VEL
LIN {X 0,Y 144.008,Z 412.231,A -85,B 0,C 180,E1 -24976.021,E2 -24976.021} C_VEL
LIN {X 0,Y 142.545,Z 408.88,A -85,B 0,C 180,E1 -24976.958,E2 -24976.958} C_VEL
LIN {X 0,Y 140.589,Z 404.469,A -85,B 0,C 180,E1 -24978.161,E2 -24978.161} C_VEL
LIN {X 0,Y 138.615,Z 400.651,A -85,B 0,C 180,E1 -24979.315,E2 -24979.315} C_VEL
LIN {X 0,Y 138.203,Z 399.015,A -85,B 0,C 180,E1 -24979.714,E2 -24979.714} C_VEL
LIN {X 0,Y 137.944,Z 397.693,A -85,B 0,C 180,E1 -24981.351,E2 -24981.351} C_VEL
LIN {X 0,Y 136.931,Z 396.051,A -85,B 0,C 180,E1 -24983.673,E2 -24983.673} C_VEL
LIN {X 0,Y 135.042,Z 394.698,A -85,B 0,C 180,E1 -24985.979,E2 -24985.979} C_VEL
LIN {X 0,Y 129.773,Z 391.444,A -85,B 0,C 180,E1 -24992.402,E2 -24992.402} C_VEL
LIN {X 0,Y 129.276,Z 390.464,A -85,B 0,C 180,E1 -24994.111,E2 -24994.111} C_VEL
LIN {X 0,Y 129.046,Z 389.415,A -85,B 0,C 180,E1 -24995.893,E2 -24995.893} C_VEL
LIN {X 0,Y 129.169,Z 389.401,A -85,B 0,C 180,E1 -25000.947,E2 -25000.947} C_VEL
LIN {X 0,Y 129.424,Z 389.364,A -85,B 0,C 180,E1 -25007.816,E2 -25007.816} C_VEL
LIN {X 0,Y 129.537,Z 389.35,A -85,B 0,C 180,E1 -25010.633,E2 -25010.633} C_VEL
LIN {X 0,Y 130.096,Z 389.265,A -85,B 0,C 180,E1 -25020.001,E2 -25020.001} C_VEL
LIN {X 0,Y 129.536,Z 389.342,A -85,B 0,C 180,E1 -25029.368,E2 -25029.368} C_VEL
LIN {X 0,Y 129.4,Z 389.361,A -85,B 0,C 180,E1 -25032.548,E2 -25032.548} C_VEL
LIN {X 0,Y 129.162,Z 389.395,A -85,B 0,C 180,E1 -25039.056,E2 -25039.056} C_VEL
LIN {X 0,Y 129.115,Z 389.385,A -85,B 0,C 180,E1 -25042.398,E2 -25042.398} C_VEL
LIN {X 0,Y 129.042,Z 389.398,A -85,B 0,C 180,E1 -25049.373,E2 -25049.373} C_VEL
LIN {X 0,Y 128.998,Z 389.413,A -85,B 0,C 180,E1 -25055.189,E2 -25055.189} C_VEL
LIN {X 0,Y 128.956,Z 389.418,A -85,B 0,C 180,E1 -25060.844,E2 -25060.844} C_VEL
LIN {X 0,Y 128.944,Z 389.432,A -85,B 0,C 180,E1 -25065.815,E2 -25065.815} C_VEL
LIN {X 0,Y 129.872,Z 392.101,A -85,B 0,C 180,E1 -25066.792,E2 -25066.792} C_VEL
LIN {X 0,Y 131.845,Z 394.665,A -85,B 0,C 180,E1 -25068.27,E2 -25068.27} C_VEL
LIN {X 0,Y 132.953,Z 396.93,A -85,B 0,C 180,E1 -25069.269,E2 -25069.269} C_VEL
LIN {X 0,Y 134.212,Z 398.513,A -85,B 0,C 180,E1 -25070.182,E2 -25070.182} C_VEL
LIN {X 0,Y 138.696,Z 407.506,A -85,B 0,C 180,E1 -25074.171,E2 -25074.171} C_VEL
LIN {X 0,Y 141.77,Z 415.334,A -85,B 0,C 180,E1 -25077.433,E2 -25077.433} C_VEL
LIN {X 0,Y 144.326,Z 423.643,A -85,B 0,C 180,E1 -25080.857,E2 -25080.857} C_VEL
LIN {X 0,Y 145.965,Z 431.969,A -85,B 0,C 180,E1 -25084.318,E2 -25084.318} C_VEL
LIN {X 0,Y 142.63,Z 441.681,A -85,B 0,C 180,E1 -25087.548,E2 -25087.548} C_VEL
LIN {X 0,Y 138.898,Z 451.144,A -85,B 0,C 180,E1 -25091.562,E2 -25091.562} C_VEL
LIN {X 0,Y 135.677,Z 458.688,A -85,B 0,C 180,E1 -25095.754,E2 -25095.754} C_VEL
LIN {X 0,Y 132.82,Z 465.638,A -85,B 0,C 180,E1 -25100.864,E2 -25100.864} C_VEL
LIN {X 0,Y 130.975,Z 470.28,A -85,B 0,C 180,E1 -25105.381,E2 -25105.381} C_VEL
LIN {X 0,Y 129.631,Z 473.861,A -85,B 0,C 180,E1 -25109.998,E2 -25109.998} C_VEL
LIN {X 0,Y 129.186,Z 475.698,A -85,B 0,C 180,E1 -25113.116,E2 -25113.116} C_VEL
LIN {X 0,Y 129.184,Z 477.065,A -85,B 0,C 180,E1 -25116.244,E2 -25116.244} C_VEL
LIN {X 0,Y 129.697,Z 478.703,A -85,B 0,C 180,E1 -25122.516,E2 -25122.516} C_VEL
LIN {X 0,Y 130.346,Z 478.937,A -85,B 0,C 180,E1 -25125.638,E2 -25125.638} C_VEL
LIN {X 0,Y 132.578,Z 478.189,A -85,B 0,C 180,E1 -25131.779,E2 -25131.779} C_VEL
LIN {X 0,Y 134.169,Z 477.236,A -85,B 0,C 180,E1 -25134.772,E2 -25134.772} C_VEL
LIN {X 0,Y 137.742,Z 474.514,A -85,B 0,C 180,E1 -25139.841,E2 -25139.841} C_VEL
LIN {X 0,Y 142.089,Z 470.418,A -85,B 0,C 180,E1 -25144.665,E2 -25144.665} C_VEL
LIN {X 0,Y 146.457,Z 465.689,A -85,B 0,C 180,E1 -25148.594,E2 -25148.594} C_VEL
LIN {X 0,Y 151.316,Z 459.816,A -85,B 0,C 180,E1 -25152.206,E2 -25152.206} C_VEL
LIN {X 0,Y 156.927,Z 452.096,A -85,B 0,C 180,E1 -25155.769,E2 -25155.769} C_VEL
LIN {X 0,Y 157.358,Z 451.058,A -85,B 0,C 180,E1 -25156.27,E2 -25156.27} C_VEL
LIN {X 0,Y 157.159,Z 445.372,A -85,B 0,C 180,E1 -25160.032,E2 -25160.032} C_VEL
LIN {X 0,Y 156.418,Z 438.827,A -85,B 0,C 180,E1 -25164.26,E2 -25164.26} C_VEL
LIN {X 0,Y 155.004,Z 432.441,A -85,B 0,C 180,E1 -25168.573,E2 -25168.573} C_VEL
LIN {X 0,Y 153.289,Z 426.842,A -85,B 0,C 180,E1 -25172.71,E2 -25172.71} C_VEL
LIN {X 0,Y 151.394,Z 421.999,A -85,B 0,C 180,E1 -25176.759,E2 -25176.759} C_VEL
LIN {X 0,Y 149.533,Z 417.863,A -85,B 0,C 180,E1 -25180.791,E2 -25180.791} C_VEL
LIN {X 0,Y 148.401,Z 415.476,A -85,B 0,C 180,E1 -25183.491,E2 -25183.491} C_VEL
LIN {X 0,Y 147.43,Z 413.176,A -85,B 0,C 180,E1 -25186.21,E2 -25186.21} C_VEL
LIN {X 0,Y 146.472,Z 411.491,A -85,B 0,C 180,E1 -25188.934,E2 -25188.934} C_VEL
LIN {X 0,Y 144.992,Z 407.09,A -85,B 0,C 180,E1 -25197.221,E2 -25197.221} C_VEL
LIN {X 0,Y 144.702,Z 406.824,A -85,B 0,C 180,E1 -25199.999,E2 -25199.999} C_VEL
LIN {X 0,Y 144.522,Z 407.26,A -85,B 0,C 180,E1 -25202.787,E2 -25202.787} C_VEL
LIN {X 0,Y 144.859,Z 409.178,A -85,B 0,C 180,E1 -25208.368,E2 -25208.368} C_VEL
LIN {X 0,Y 145.423,Z 410.488,A -85,B 0,C 180,E1 -25211.146,E2 -25211.146} C_VEL
LIN {X 0,Y 148.496,Z 419.572,A -85,B 0,C 180,E1 -25220.79,E2 -25220.79} C_VEL
LIN {X 0,Y 151.1,Z 426.989,A -85,B 0,C 180,E1 -25226.222,E2 -25226.222} C_VEL
LIN {X 0,Y 152.872,Z 432.518,A -85,B 0,C 180,E1 -25229.608,E2 -25229.608} C_VEL
LIN {X 0,Y 154.909,Z 440.365,A -85,B 0,C 180,E1 -25233.764,E2 -25233.764} C_VEL
LIN {X 0,Y 156.658,Z 449.53,A -85,B 0,C 180,E1 -25238.086,E2 -25238.086} C_VEL
LIN {X 0,Y 156.174,Z 453.647,A -85,B 0,C 180,E1 -25239.477,E2 -25239.477} C_VEL
LIN {X 0,Y 153.862,Z 464.134,A -85,B 0,C 180,E1 -25243.046,E2 -25243.046} C_VEL
LIN {X 0,Y 150.888,Z 473.528,A -85,B 0,C 180,E1 -25246.608,E2 -25246.608} C_VEL
LIN {X 0,Y 147.555,Z 481.827,A -85,B 0,C 180,E1 -25250.274,E2 -25250.274} C_VEL
LIN {X 0,Y 144.516,Z 487.957,A -85,B 0,C 180,E1 -25253.437,E2 -25253.437} C_VEL
LIN {X 0,Y 140.597,Z 493.406,A -85,B 0,C 180,E1 -25256.645,E2 -25256.645} C_VEL
LIN {X 0,Y 136.257,Z 498.733,A -85,B 0,C 180,E1 -25260.662,E2 -25260.662} C_VEL
LIN {X 0,Y 132.772,Z 502.948,A -85,B 0,C 180,E1 -25264.949,E2 -25264.949} C_VEL
LIN {X 0,Y 130.904,Z 505.171,A -85,B 0,C 180,E1 -25267.928,E2 -25267.928} C_VEL
LIN {X 0,Y 128.36,Z 508.402,A -85,B 0,C 180,E1 -25274.114,E2 -25274.114} C_VEL
LIN {X 0,Y 127.749,Z 509.443,A -85,B 0,C 180,E1 -25277.29,E2 -25277.29} C_VEL
LIN {X 0,Y 127.726,Z 510.297,A -85,B 0,C 180,E1 -25283.684,E2 -25283.684} C_VEL
LIN {X 0,Y 128.196,Z 510.145,A -85,B 0,C 180,E1 -25286.86,E2 -25286.86} C_VEL
LIN {X 0,Y 128.595,Z 509.556,A -85,B 0,C 180,E1 -25290.002,E2 -25290.002} C_VEL
LIN {X 0,Y 128.173,Z 508.379,A -85,B 0,C 180,E1 -25293.146,E2 -25293.146} C_VEL
LIN {X 0,Y 127.695,Z 505.811,A -85,B 0,C 180,E1 -25297.834,E2 -25297.834} C_VEL
LIN {X 0,Y 127.867,Z 502.079,A -85,B 0,C 180,E1 -25302.703,E2 -25302.703} C_VEL
LIN {X 0,Y 128.869,Z 497.27,A -85,B 0,C 180,E1 -25307.457,E2 -25307.457} C_VEL
LIN {X 0,Y 131.124,Z 490.04,A -85,B 0,C 180,E1 -25312.869,E2 -25312.869} C_VEL
LIN {X 0,Y 134.219,Z 482.014,A -85,B 0,C 180,E1 -25317.423,E2 -25317.423} C_VEL
LIN {X 0,Y 136.351,Z 472.186,A -85,B 0,C 180,E1 -25321.895,E2 -25321.895} C_VEL
LIN {X 0,Y 138.387,Z 462.638,A -85,B 0,C 180,E1 -25325.38,E2 -25325.38} C_VEL
LIN {X 0,Y 140.101,Z 451.256,A -85,B 0,C 180,E1 -25328.835,E2 -25328.835} C_VEL
LIN {X 0,Y 141.035,Z 439.657,A -85,B 0,C 180,E1 -25331.787,E2 -25331.787} C_VEL
LIN {X 0,Y 141.042,Z 428.823,A -85,B 0,C 180,E1 -25334.238,E2 -25334.238} C_VEL
LIN {X 0,Y 140.406,Z 420.518,A -85,B 0,C 180,E1 -25336.012,E2 -25336.012} C_VEL
LIN {X 0,Y 137.932,Z 413.57,A -85,B 0,C 180,E1 -25338.03,E2 -25338.03} C_VEL
LIN {X 0,Y 135.611,Z 408.332,A -85,B 0,C 180,E1 -25339.683,E2 -25339.683} C_VEL
LIN {X 0,Y 133.854,Z 404.182,A -85,B 0,C 180,E1 -25340.946,E2 -25340.946} C_VEL
LIN {X 0,Y 131.433,Z 399.969,A -85,B 0,C 180,E1 -25342.538,E2 -25342.538} C_VEL
LIN {X 0,Y 130.738,Z 397.768,A -85,B 0,C 180,E1 -25343.151,E2 -25343.151} C_VEL
LIN {X 0,Y 130.204,Z 394.822,A -85,B 0,C 180,E1 -25347.333,E2 -25347.333} C_VEL
LIN {X 0,Y 129.501,Z 391.431,A -85,B 0,C 180,E1 -25352.53,E2 -25352.53} C_VEL
LIN {X 0,Y 129.276,Z 390.464,A -85,B 0,C 180,E1 -25354.111,E2 -25354.111} C_VEL
LIN {X 0,Y 128.817,Z 389.762,A -85,B 0,C 180,E1 -25355.803,E2 -25355.803} C_VEL
LIN {X 0,Y 127.41,Z 389.619,A -85,B 0,C 180,E1 -25358.364,E2 -25358.364} C_VEL
LIN {X 0,Y 122.629,Z 390.223,A -85,B 0,C 180,E1 -25366.373,E2 -25366.373} C_VEL
LIN {X 0,Y 122.372,Z 390.239,A -85,B 0,C 180,E1 -25368.259,E2 -25368.259} C_VEL
LIN {X 0,Y 122.462,Z 390.23,A -85,B 0,C 180,E1 -25373.41,E2 -25373.41} C_VEL
LIN {X 0,Y 123.05,Z 390.142,A -85,B 0,C 180,E1 -25380.001,E2 -25380.001} C_VEL
LIN {X 0,Y 122.429,Z 390.212,A -85,B 0,C 180,E1 -25387.205,E2 -25387.205} C_VEL
LIN {X 0,Y 122.371,Z 390.237,A -85,B 0,C 180,E1 -25392.477,E2 -25392.477} C_VEL
LIN {X 0,Y 122.053,Z 390.278,A -85,B 0,C 180,E1 -25400.213,E2 -25400.213} C_VEL
LIN {X 0,Y 121.99,Z 390.273,A -85,B 0,C 180,E1 -25403.784,E2 -25403.784} C_VEL
LIN {X 0,Y 121.948,Z 390.279,A -85,B 0,C 180,E1 -25410.173,E2 -25410.173} C_VEL
LIN {X 0,Y 121.918,Z 390.296,A -85,B 0,C 180,E1 -25416.189,E2 -25416.189} C_VEL
LIN {X 0,Y 121.871,Z 390.302,A -85,B 0,C 180,E1 -25421.815,E2 -25421.815} C_VEL
LIN {X 0,Y 122.616,Z 392.788,A -85,B 0,C 180,E1 -25422.799,E2 -25422.799} C_VEL
LIN {X 0,Y 124.548,Z 395.025,A -85,B 0,C 180,E1 -25424.467,E2 -25424.467} C_VEL
LIN {X 0,Y 128.075,Z 401.057,A -85,B 0,C 180,E1 -25427.801,E2 -25427.801} C_VEL
LIN {X 0,Y 130.421,Z 405.295,A -85,B 0,C 180,E1 -25430.045,E2 -25430.045} C_VEL
LIN {X 0,Y 133.824,Z 412.609,A -85,B 0,C 180,E1 -25433.614,E2 -25433.614} C_VEL
LIN {X 0,Y 136.257,Z 419.417,A -85,B 0,C 180,E1 -25436.688,E2 -25436.688} C_VEL
LIN {X 0,Y 138.513,Z 427.667,A -85,B 0,C 180,E1 -25440.396,E2 -25440.396} C_VEL
LIN {X 0,Y 139.554,Z 433.508,A -85,B 0,C 180,E1 -25443.046,E2 -25443.046} C_VEL
LIN {X 0,Y 137.569,Z 439.477,A -85,B 0,C 180,E1 -25445.07,E2 -25445.07} C_VEL
LIN {X 0,Y 134.175,Z 448.025,A -85,B 0,C 180,E1 -25448.488,E2 -25448.488} C_VEL
LIN {X 0,Y 130.517,Z 456.351,A -85,B 0,C 180,E1 -25452.771,E2 -25452.771} C_VEL
LIN {X 0,Y 127.531,Z 463.044,A -85,B 0,C 180,E1 -25457.263,E2 -25457.263} C_VEL
LIN {X 0,Y 125.186,Z 468.408,A -85,B 0,C 180,E1 -25461.929,E2 -25461.929} C_VEL
LIN {X 0,Y 123.409,Z 472.634,A -85,B 0,C 180,E1 -25466.733,E2 -25466.733} C_VEL
LIN {X 0,Y 122.553,Z 474.896,A -85,B 0,C 180,E1 -25469.998,E2 -25469.998} C_VEL
LIN {X 0,Y 122.126,Z 476.682,A -85,B 0,C 180,E1 -25473.297,E2 -25473.297} C_VEL
LIN {X 0,Y 122.137,Z 478.026,A -85,B 0,C 180,E1 -25476.606,E2 -25476.606} C_VEL
LIN {X 0,Y 122.776,Z 479.627,A -85,B 0,C 180,E1 -25483.311,E2 -25483.311} C_VEL
LIN {X 0,Y 124.588,Z 479.596,A -85,B 0,C 180,E1 -25489.781,E2 -25489.781} C_VEL
LIN {X 0,Y 127.719,Z 478.029,A -85,B 0,C 180,E1 -25496.115,E2 -25496.115} C_VEL
LIN {X 0,Y 131.389,Z 475.405,A -85,B 0,C 180,E1 -25501.145,E2 -25501.145} C_VEL
LIN {X 0,Y 136.263,Z 471.085,A -85,B 0,C 180,E1 -25506.377,E2 -25506.377} C_VEL
LIN {X 0,Y 140.933,Z 466.297,A -85,B 0,C 180,E1 -25510.409,E2 -25510.409} C_VEL
LIN {X 0,Y 146.033,Z 460.426,A -85,B 0,C 180,E1 -25514.058,E2 -25514.058} C_VEL
LIN {X 0,Y 151.025,Z 453.927,A -85,B 0,C 180,E1 -25517.13,E2 -25517.13} C_VEL
LIN {X 0,Y 151.289,Z 450.645,A -85,B 0,C 180,E1 -25519.43,E2 -25519.43} C_VEL
LIN {X 0,Y 151.049,Z 444.68,A -85,B 0,C 180,E1 -25523.656,E2 -25523.656} C_VEL
LIN {X 0,Y 150.425,Z 439.749,A -85,B 0,C 180,E1 -25527.24,E2 -25527.24} C_VEL
LIN {X 0,Y 149.133,Z 433.692,A -85,B 0,C 180,E1 -25531.883,E2 -25531.883} C_VEL
LIN {X 0,Y 147.703,Z 428.741,A -85,B 0,C 180,E1 -25536.143,E2 -25536.143} C_VEL
LIN {X 0,Y 146.131,Z 424.628,A -85,B 0,C 180,E1 -25540.326,E2 -25540.326} C_VEL
LIN {X 0,Y 145.216,Z 422.127,A -85,B 0,C 180,E1 -25543.118,E2 -25543.118} C_VEL
LIN {X 0,Y 143.602,Z 418.199,A -85,B 0,C 180,E1 -25548.71,E2 -25548.71} C_VEL
LIN {X 0,Y 142.486,Z 413.915,A -85,B 0,C 180,E1 -25557.172,E2 -25557.172} C_VEL
LIN {X 0,Y 142.305,Z 413.511,A -85,B 0,C 180,E1 -25559.999,E2 -25559.999} C_VEL
LIN {X 0,Y 142.123,Z 414.018,A -85,B 0,C 180,E1 -25562.834,E2 -25562.834} C_VEL
LIN {X 0,Y 142.69,Z 416.653,A -85,B 0,C 180,E1 -25569.925,E2 -25569.925} C_VEL
LIN {X 0,Y 142.911,Z 417.583,A -85,B 0,C 180,E1 -25571.344,E2 -25571.344} C_VEL
LIN {X 0,Y 145.095,Z 425.337,A -85,B 0,C 180,E1 -25579.819,E2 -25579.819} C_VEL
LIN {X 0,Y 147.205,Z 432.621,A -85,B 0,C 180,E1 -25585.447,E2 -25585.447} C_VEL
LIN {X 0,Y 148.575,Z 437.84,A -85,B 0,C 180,E1 -25588.836,E2 -25588.836} C_VEL
LIN {X 0,Y 149.899,Z 444.182,A -85,B 0,C 180,E1 -25592.446,E2 -25592.446} C_VEL
LIN {X 0,Y 151.112,Z 452.094,A -85,B 0,C 180,E1 -25596.517,E2 -25596.517} C_VEL
LIN {X 0,Y 151.21,Z 453.457,A -85,B 0,C 180,E1 -25597.172,E2 -25597.172} C_VEL
LIN {X 0,Y 148.936,Z 462.729,A -85,B 0,C 180,E1 -25600.462,E2 -25600.462} C_VEL
LIN {X 0,Y 146.135,Z 471.349,A -85,B 0,C 180,E1 -25603.834,E2 -25603.834} C_VEL
LIN {X 0,Y 142.513,Z 479.992,A -85,B 0,C 180,E1 -25607.707,E2 -25607.707} C_VEL
LIN {X 0,Y 138.707,Z 487.35,A -85,B 0,C 180,E1 -25611.637,E2 -25611.637} C_VEL
LIN {X 0,Y 135.516,Z 491.75,A -85,B 0,C 180,E1 -25614.31,E2 -25614.31} C_VEL
LIN {X 0,Y 130.065,Z 498.039,A -85,B 0,C 180,E1 -25619.117,E2 -25619.117} C_VEL
LIN {X 0,Y 126.316,Z 502.209,A -85,B 0,C 180,E1 -25623.572,E2 -25623.572} C_VEL
LIN {X 0,Y 122.66,Z 506.186,A -85,B 0,C 180,E1 -25629.895,E2 -25629.895} C_VEL
LIN {X 0,Y 120.794,Z 508.596,A -85,B 0,C 180,E1 -25636.545,E2 -25636.545} C_VEL
LIN {X 0,Y 120.652,Z 509.406,A -85,B 0,C 180,E1 -25643.312,E2 -25643.312} C_VEL
LIN {X 0,Y 121.094,Z 509.234,A -85,B 0,C 180,E1 -25646.675,E2 -25646.675} C_VEL
LIN {X 0,Y 121.537,Z 508.627,A -85,B 0,C 180,E1 -25650.002,E2 -25650.002} C_VEL
LIN {X 0,Y 121.063,Z 507.404,A -85,B 0,C 180,E1 -25653.33,E2 -25653.33} C_VEL
LIN {X 0,Y 120.621,Z 505.043,A -85,B 0,C 180,E1 -25657.903,E2 -25657.903} C_VEL
LIN {X 0,Y 120.892,Z 501.009,A -85,B 0,C 180,E1 -25663.449,E2 -25663.449} C_VEL
LIN {X 0,Y 122.028,Z 496.145,A -85,B 0,C 180,E1 -25668.47,E2 -25668.47} C_VEL
LIN {X 0,Y 124.081,Z 490.011,A -85,B 0,C 180,E1 -25673.361,E2 -25673.361} C_VEL
LIN {X 0,Y 127.139,Z 482.768,A -85,B 0,C 180,E1 -25677.817,E2 -25677.817} C_VEL
LIN {X 0,Y 129.178,Z 474.44,A -85,B 0,C 180,E1 -25682.039,E2 -25682.039} C_VEL
LIN {X 0,Y 131.543,Z 464.733,A -85,B 0,C 180,E1 -25685.997,E2 -25685.997} C_VEL
LIN {X 0,Y 133.327,Z 455.133,A -85,B 0,C 180,E1 -25689.241,E2 -25689.241} C_VEL
LIN {X 0,Y 134.7,Z 444.407,A -85,B 0,C 180,E1 -25692.313,E2 -25692.313} C_VEL
LIN {X 0,Y 135.245,Z 432.88,A -85,B 0,C 180,E1 -25695.215,E2 -25695.215} C_VEL
LIN {X 0,Y 134.932,Z 423.65,A -85,B 0,C 180,E1 -25697.382,E2 -25697.382} C_VEL
LIN {X 0,Y 133.501,Z 418.92,A -85,B 0,C 180,E1 -25698.849,E2 -25698.849} C_VEL
LIN {X 0,Y 128.951,Z 408.029,A -85,B 0,C 180,E1 -25702.676,E2 -25702.676} C_VEL
LIN {X 0,Y 126.903,Z 403.719,A -85,B 0,C 180,E1 -25704.326,E2 -25704.326} C_VEL
LIN {X 0,Y 126.098,Z 402.216,A -85,B 0,C 180,E1 -25704.955,E2 -25704.955} C_VEL
LIN {X 0,Y 123.909,Z 398.464,A -85,B 0,C 180,E1 -25706.671,E2 -25706.671} C_VEL
LIN {X 0,Y 123.293,Z 396.438,A -85,B 0,C 180,E1 -25707.337,E2 -25707.337} C_VEL
LIN {X 0,Y 122.612,Z 393.12,A -85,B 0,C 180,E1 -25712.707,E2 -25712.707} C_VEL
LIN {X 0,Y 122.075,Z 390.284,A -85,B 0,C 180,E1 -25717.972,E2 -25717.972} C_VEL
LIN {X 0,Y 122.127,Z 390.278,A -85,B 0,C 180,E1 -25723.278,E2 -25723.278} C_VEL
LIN {X 0,Y 122.372,Z 390.239,A -85,B 0,C 180,E1 -25728.259,E2 -25728.259} C_VEL
LIN {X 0,Y 121.795,Z 390.315,A -85,B 0,C 180,E1 -25731.011,E2 -25731.011} C_VEL
LIN {X 0,Y 120.357,Z 390.492,A -85,B 0,C 180,E1 -25733.735,E2 -25733.735} C_VEL
LIN {X 0,Y 115.98,Z 391.032,A -85,B 0,C 180,E1 -25741.257,E2 -25741.257} C_VEL
LIN {X 0,Y 115.56,Z 391.085,A -85,B 0,C 180,E1 -25743.245,E2 -25743.245} C_VEL
LIN {X 0,Y 115.399,Z 391.109,A -85,B 0,C 180,E1 -25750.528,E2 -25750.528} C_VEL
LIN {X 0,Y 115.152,Z 391.122,A -85,B 0,C 180,E1 -25754.131,E2 -25754.131} C_VEL
LIN {X 0,Y 114.986,Z 391.148,A -85,B 0,C 180,E1 -25761.515,E2 -25761.515} C_VEL
LIN {X 0,Y 114.877,Z 391.169,A -85,B 0,C 180,E1 -25765.358,E2 -25765.358} C_VEL
LIN {X 0,Y 114.875,Z 391.161,A -85,B 0,C 180,E1 -25771.068,E2 -25771.068} C_VEL
LIN {X 0,Y 114.866,Z 391.265,A -85,B 0,C 180,E1 -25776.877,E2 -25776.877} C_VEL
LIN {X 0,Y 115.661,Z 393.74,A -85,B 0,C 180,E1 -25778.108,E2 -25778.108} C_VEL
LIN {X 0,Y 118.159,Z 396.603,A -85,B 0,C 180,E1 -25780.725,E2 -25780.725} C_VEL
LIN {X 0,Y 119.553,Z 399.462,A -85,B 0,C 180,E1 -25782.441,E2 -25782.441} C_VEL
LIN {X 0,Y 121.206,Z 401.666,A -85,B 0,C 180,E1 -25784.093,E2 -25784.093} C_VEL
LIN {X 0,Y 125.766,Z 410.282,A -85,B 0,C 180,E1 -25789.196,E2 -25789.196} C_VEL
LIN {X 0,Y 128.894,Z 417.762,A -85,B 0,C 180,E1 -25793.143,E2 -25793.143} C_VEL
LIN {X 0,Y 131.315,Z 425.626,A -85,B 0,C 180,E1 -25797.021,E2 -25797.021} C_VEL
LIN {X 0,Y 132.652,Z 431.84,A -85,B 0,C 180,E1 -25800.049,E2 -25800.049} C_VEL
LIN {X 0,Y 133.163,Z 436.016,A -85,B 0,C 180,E1 -25802.067,E2 -25802.067} C_VEL
LIN {X 0,Y 129.767,Z 444.486,A -85,B 0,C 180,E1 -25805.18,E2 -25805.18} C_VEL
LIN {X 0,Y 126.309,Z 452.308,A -85,B 0,C 180,E1 -25808.795,E2 -25808.795} C_VEL
LIN {X 0,Y 122.62,Z 459.994,A -85,B 0,C 180,E1 -25813.344,E2 -25813.344} C_VEL
LIN {X 0,Y 119.738,Z 466.131,A -85,B 0,C 180,E1 -25818.143,E2 -25818.143} C_VEL
LIN {X 0,Y 117.532,Z 471.028,A -85,B 0,C 180,E1 -25823.129,E2 -25823.129} C_VEL
LIN {X 0,Y 115.877,Z 474.853,A -85,B 0,C 180,E1 -25828.26,E2 -25828.26} C_VEL
LIN {X 0,Y 115.065,Z 477.664,A -85,B 0,C 180,E1 -25833.499,E2 -25833.499} C_VEL
LIN {X 0,Y 115.099,Z 478.987,A -85,B 0,C 180,E1 -25837.012,E2 -25837.012} C_VEL
LIN {X 0,Y 115.804,Z 480.498,A -85,B 0,C 180,E1 -25843.823,E2 -25843.823} C_VEL
LIN {X 0,Y 116.695,Z 480.672,A -85,B 0,C 180,E1 -25847.523,E2 -25847.523} C_VEL
LIN {X 0,Y 119.445,Z 479.83,A -85,B 0,C 180,E1 -25854.32,E2 -25854.32} C_VEL
LIN {X 0,Y 121.345,Z 478.81,A -85,B 0,C 180,E1 -25857.6,E2 -25857.6} C_VEL
LIN {X 0,Y 125.115,Z 476.294,A -85,B 0,C 180,E1 -25862.584,E2 -25862.584} C_VEL
LIN {X 0,Y 130.579,Z 471.751,A -85,B 0,C 180,E1 -25868.237,E2 -25868.237} C_VEL
LIN {X 0,Y 135.562,Z 466.905,A -85,B 0,C 180,E1 -25872.371,E2 -25872.371} C_VEL
LIN {X 0,Y 140.97,Z 460.971,A -85,B 0,C 180,E1 -25876.084,E2 -25876.084} C_VEL
LIN {X 0,Y 145.087,Z 455.753,A -85,B 0,C 180,E1 -25878.658,E2 -25878.658} C_VEL
LIN {X 0,Y 145.342,Z 450.483,A -85,B 0,C 180,E1 -25882.811,E2 -25882.811} C_VEL
LIN {X 0,Y 145.136,Z 445.096,A -85,B 0,C 180,E1 -25887.031,E2 -25887.031} C_VEL
LIN {X 0,Y 144.502,Z 440.149,A -85,B 0,C 180,E1 -25891.094,E2 -25891.094} C_VEL
LIN {X 0,Y 143.462,Z 435.439,A -85,B 0,C 180,E1 -25895.391,E2 -25895.391} C_VEL
LIN {X 0,Y 142.347,Z 431.147,A -85,B 0,C 180,E1 -25899.78,E2 -25899.78} C_VEL
LIN {X 0,Y 141.224,Z 427.645,A -85,B 0,C 180,E1 -25904.114,E2 -25904.114} C_VEL
LIN {X 0,Y 140.343,Z 424.694,A -85,B 0,C 180,E1 -25908.444,E2 -25908.444} C_VEL
LIN {X 0,Y 139.609,Z 420.573,A -85,B 0,C 180,E1 -25917.114,E2 -25917.114} C_VEL
LIN {X 0,Y 139.543,Z 420.078,A -85,B 0,C 180,E1 -25919.999,E2 -25919.999} C_VEL
LIN {X 0,Y 139.368,Z 420.625,A -85,B 0,C 180,E1 -25922.89,E2 -25922.89} C_VEL
LIN {X 0,Y 139.686,Z 422.667,A -85,B 0,C 180,E1 -25928.681,E2 -25928.681} C_VEL
LIN {X 0,Y 139.868,Z 423.452,A -85,B 0,C 180,E1 -25930.127,E2 -25930.127} C_VEL
LIN {X 0,Y 140.971,Z 429.681,A -85,B 0,C 180,E1 -25937.404,E2 -25937.404} C_VEL
LIN {X 0,Y 141.524,Z 431.602,A -85,B 0,C 180,E1 -25939.353,E2 -25939.353} C_VEL
LIN {X 0,Y 142.963,Z 437.66,A -85,B 0,C 180,E1 -25944.369,E2 -25944.369} C_VEL
LIN {X 0,Y 143.95,Z 442.294,A -85,B 0,C 180,E1 -25947.634,E2 -25947.634} C_VEL
LIN {X 0,Y 144.906,Z 448.469,A -85,B 0,C 180,E1 -25951.424,E2 -25951.424} C_VEL
LIN {X 0,Y 145.632,Z 455.572,A -85,B 0,C 180,E1 -25955.387,E2 -25955.387} C_VEL
LIN {X 0,Y 145.623,Z 456.768,A -85,B 0,C 180,E1 -25955.979,E2 -25955.979} C_VEL
LIN {X 0,Y 142.521,Z 466.762,A -85,B 0,C 180,E1 -25959.87,E2 -25959.87} C_VEL
LIN {X 0,Y 138.788,Z 475.806,A -85,B 0,C 180,E1 -25963.817,E2 -25963.817} C_VEL
LIN {X 0,Y 135.195,Z 482.998,A -85,B 0,C 180,E1 -25967.487,E2 -25967.487} C_VEL
LIN {X 0,Y 131.514,Z 489.044,A -85,B 0,C 180,E1 -25971.107,E2 -25971.107} C_VEL
LIN {X 0,Y 125.543,Z 495.717,A -85,B 0,C 180,E1 -25975.96,E2 -25975.96} C_VEL
LIN {X 0,Y 121.248,Z 500.125,A -85,B 0,C 180,E1 -25980.395,E2 -25980.395} C_VEL
LIN {X 0,Y 117.743,Z 503.629,A -85,B 0,C 180,E1 -25985.305,E2 -25985.305} C_VEL
LIN {X 0,Y 114.679,Z 506.779,A -85,B 0,C 180,E1 -25992.159,E2 -25992.159} C_VEL
LIN {X 0,Y 113.463,Z 508.312,A -85,B 0,C 180,E1 -25999.293,E2 -25999.293} C_VEL
LIN {X 0,Y 113.605,Z 508.517,A -85,B 0,C 180,E1 -26002.895,E2 -26002.895} C_VEL
LIN {X 0,Y 113.998,Z 508.323,A -85,B 0,C 180,E1 -26006.468,E2 -26006.468} C_VEL
LIN {X 0,Y 114.475,Z 507.689,A -85,B 0,C 180,E1 -26010.003,E2 -26010.003} C_VEL
LIN {X 0,Y 113.958,Z 506.43,A -85,B 0,C 180,E1 -26013.538,E2 -26013.538} C_VEL
LIN {X 0,Y 113.56,Z 504.243,A -85,B 0,C 180,E1 -26018.029,E2 -26018.029} C_VEL
LIN {X 0,Y 113.915,Z 499.934,A -85,B 0,C 180,E1 -26024.29,E2 -26024.29} C_VEL
LIN {X 0,Y 115.245,Z 495.02,A -85,B 0,C 180,E1 -26029.6,E2 -26029.6} C_VEL
LIN {X 0,Y 117.556,Z 488.834,A -85,B 0,C 180,E1 -26034.742,E2 -26034.742} C_VEL
LIN {X 0,Y 120.413,Z 482.417,A -85,B 0,C 180,E1 -26038.898,E2 -26038.898} C_VEL
LIN {X 0,Y 122.935,Z 473.075,A -85,B 0,C 180,E1 -26043.878,E2 -26043.878} C_VEL
LIN {X 0,Y 125.534,Z 463.215,A -85,B 0,C 180,E1 -26048.016,E2 -26048.016} C_VEL
LIN {X 0,Y 127.657,Z 452.194,A -85,B 0,C 180,E1 -26051.827,E2 -26051.827} C_VEL
LIN {X 0,Y 128.979,Z 441.772,A -85,B 0,C 180,E1 -26054.899,E2 -26054.899} C_VEL
LIN {X 0,Y 129.517,Z 430.45,A -85,B 0,C 180,E1 -26057.874,E2 -26057.874} C_VEL
LIN {X 0,Y 129.425,Z 426.634,A -85,B 0,C 180,E1 -26058.841,E2 -26058.841} C_VEL
LIN {X 0,Y 127.049,Z 419.259,A -85,B 0,C 180,E1 -26061.514,E2 -26061.514} C_VEL
LIN {X 0,Y 124.155,Z 411.968,A -85,B 0,C 180,E1 -26064.41,E2 -26064.41} C_VEL
LIN {X 0,Y 122.13,Z 407.337,A -85,B 0,C 180,E1 -26066.367,E2 -26066.367} C_VEL
LIN {X 0,Y 119.919,Z 402.931,A -85,B 0,C 180,E1 -26068.466,E2 -26068.466} C_VEL
LIN {X 0,Y 119.344,Z 401.604,A -85,B 0,C 180,E1 -26069.045,E2 -26069.045} C_VEL
LIN {X 0,Y 116.862,Z 397.9,A -85,B 0,C 180,E1 -26071.365,E2 -26071.365} C_VEL
LIN {X 0,Y 115.732,Z 394.864,A -85,B 0,C 180,E1 -26072.662,E2 -26072.662} C_VEL
LIN {X 0,Y 115.025,Z 391.163,A -85,B 0,C 180,E1 -26079.783,E2 -26079.783} C_VEL
LIN {X 0,Y 115.323,Z 391.118,A -85,B 0,C 180,E1 -26088.338,E2 -26088.338} C_VEL
LIN {X 0,Y 115.403,Z 391.108,A -85,B 0,C 180,E1 -26093.005,E2 -26093.005} C_VEL
LIN {X 0,Y 116.002,Z 391.019,A -85,B 0,C 180,E1 -26100.001,E2 -26100.001} C_VEL
LIN {X 0,Y 115.56,Z 391.085,A -85,B 0,C 180,E1 -26103.245,E2 -26103.245} C_VEL
LIN {X 0,Y 114.721,Z 391.218,A -85,B 0,C 180,E1 -26106.152,E2 -26106.152} C_VEL
LIN {X 0,Y 113.051,Z 391.445,A -85,B 0,C 180,E1 -26109.023,E2 -26109.023} C_VEL
LIN {X 0,Y 108.321,Z 392.013,A -85,B 0,C 180,E1 -26117.004,E2 -26117.004} C_VEL
LIN {X 0,Y 107.904,Z 392.042,A -85,B 0,C 180,E1 -26119.131,E2 -26119.131} C_VEL
LIN {X 0,Y 107.864,Z 392.033,A -85,B 0,C 180,E1 -26124.184,E2 -26124.184} C_VEL
LIN {X 0,Y 107.838,Z 392.08,A -85,B 0,C 180,E1 -26130.203,E2 -26130.203} C_VEL
LIN {X 0,Y 108.768,Z 394.848,A -85,B 0,C 180,E1 -26132.072,E2 -26132.072} C_VEL
LIN {X 0,Y 111.053,Z 397.131,A -85,B 0,C 180,E1 -26135.105,E2 -26135.105} C_VEL
LIN {X 0,Y 111.527,Z 397.649,A -85,B 0,C 180,E1 -26135.702,E2 -26135.702} C_VEL
LIN {X 0,Y 112.503,Z 399.945,A -85,B 0,C 180,E1 -26137.275,E2 -26137.275} C_VEL
LIN {X 0,Y 114.699,Z 403.055,A -85,B 0,C 180,E1 -26140.045,E2 -26140.045} C_VEL
LIN {X 0,Y 118.096,Z 409.078,A -85,B 0,C 180,E1 -26144.424,E2 -26144.424} C_VEL
LIN {X 0,Y 121.377,Z 416.029,A -85,B 0,C 180,E1 -26148.829,E2 -26148.829} C_VEL
LIN {X 0,Y 124.119,Z 423.694,A -85,B 0,C 180,E1 -26153.186,E2 -26153.186} C_VEL
LIN {X 0,Y 126.174,Z 432.272,A -85,B 0,C 180,E1 -26157.774,E2 -26157.774} C_VEL
LIN {X 0,Y 126.798,Z 436.625,A -85,B 0,C 180,E1 -26160.074,E2 -26160.074} C_VEL
LIN {X 0,Y 126.595,Z 438.54,A -85,B 0,C 180,E1 -26160.935,E2 -26160.935} C_VEL
LIN {X 0,Y 122.675,Z 447.529,A -85,B 0,C 180,E1 -26164.551,E2 -26164.551} C_VEL
LIN {X 0,Y 118.41,Z 456.317,A -85,B 0,C 180,E1 -26169.135,E2 -26169.135} C_VEL
LIN {X 0,Y 114.834,Z 463.392,A -85,B 0,C 180,E1 -26174.011,E2 -26174.011} C_VEL
LIN {X 0,Y 112.029,Z 469.033,A -85,B 0,C 180,E1 -26179.149,E2 -26179.149} C_VEL
LIN {X 0,Y 109.883,Z 473.505,A -85,B 0,C 180,E1 -26184.492,E2 -26184.492} C_VEL
LIN {X 0,Y 108.399,Z 476.944,A -85,B 0,C 180,E1 -26189.997,E2 -26189.997} C_VEL
LIN {X 0,Y 108.053,Z 479.949,A -85,B 0,C 180,E1 -26197.472,E2 -26197.472} C_VEL
LIN {X 0,Y 108.833,Z 481.367,A -85,B 0,C 180,E1 -26204.383,E2 -26204.383} C_VEL
LIN {X 0,Y 109.906,Z 481.542,A -85,B 0,C 180,E1 -26208.644,E2 -26208.644} C_VEL
LIN {X 0,Y 112.991,Z 480.65,A -85,B 0,C 180,E1 -26215.808,E2 -26215.808} C_VEL
LIN {X 0,Y 115.062,Z 479.583,A -85,B 0,C 180,E1 -26219.248,E2 -26219.248} C_VEL
LIN {X 0,Y 118.941,Z 477.178,A -85,B 0,C 180,E1 -26224.182,E2 -26224.182} C_VEL
LIN {X 0,Y 123.395,Z 473.806,A -85,B 0,C 180,E1 -26228.79,E2 -26228.79} C_VEL
LIN {X 0,Y 128.534,Z 469.29,A -85,B 0,C 180,E1 -26233.113,E2 -26233.113} C_VEL
LIN {X 0,Y 135.179,Z 462.513,A -85,B 0,C 180,E1 -26237.69,E2 -26237.69} C_VEL
LIN {X 0,Y 138.419,Z 458.849,A -85,B 0,C 180,E1 -26239.602,E2 -26239.602} C_VEL
LIN {X 0,Y 139.072,Z 457.823,A -85,B 0,C 180,E1 -26240.209,E2 -26240.209} C_VEL
LIN {X 0,Y 139.558,Z 452.259,A -85,B 0,C 180,E1 -26245.017,E2 -26245.017} C_VEL
LIN {X 0,Y 139.46,Z 446.862,A -85,B 0,C 180,E1 -26249.738,E2 -26249.738} C_VEL
LIN {X 0,Y 138.913,Z 441.823,A -85,B 0,C 180,E1 -26254.531,E2 -26254.531} C_VEL
LIN {X 0,Y 138.117,Z 437.552,A -85,B 0,C 180,E1 -26259.133,E2 -26259.133} C_VEL
LIN {X 0,Y 137.074,Z 432.998,A -85,B 0,C 180,E1 -26265.145,E2 -26265.145} C_VEL
LIN {X 0,Y 136.665,Z 431.13,A -85,B 0,C 180,E1 -26268.129,E2 -26268.129} C_VEL
LIN {X 0,Y 136.316,Z 427.053,A -85,B 0,C 180,E1 -26277.044,E2 -26277.044} C_VEL
LIN {X 0,Y 136.425,Z 426.483,A -85,B 0,C 180,E1 -26279.999,E2 -26279.999} C_VEL
LIN {X 0,Y 136.258,Z 427.073,A -85,B 0,C 180,E1 -26282.956,E2 -26282.956} C_VEL
LIN {X 0,Y 136.524,Z 429.236,A -85,B 0,C 180,E1 -26288.883,E2 -26288.883} C_VEL
LIN {X 0,Y 137.141,Z 435.199,A -85,B 0,C 180,E1 -26296.37,E2 -26296.37} C_VEL
LIN {X 0,Y 137.734,Z 438.791,A -85,B 0,C 180,E1 -26299.908,E2 -26299.908} C_VEL
LIN {X 0,Y 138.713,Z 443.787,A -85,B 0,C 180,E1 -26304.224,E2 -26304.224} C_VEL
LIN {X 0,Y 139.408,Z 448.811,A -85,B 0,C 180,E1 -26307.87,E2 -26307.87} C_VEL
LIN {X 0,Y 139.971,Z 455.936,A -85,B 0,C 180,E1 -26312.42,E2 -26312.42} C_VEL
LIN {X 0,Y 140.079,Z 459.192,A -85,B 0,C 180,E1 -26314.362,E2 -26314.362} C_VEL
LIN {X 0,Y 138.318,Z 464.576,A -85,B 0,C 180,E1 -26316.615,E2 -26316.615} C_VEL
LIN {X 0,Y 135.203,Z 472.086,A -85,B 0,C 180,E1 -26319.943,E2 -26319.943} C_VEL
LIN {X 0,Y 130.733,Z 480.815,A -85,B 0,C 180,E1 -26324.335,E2 -26324.335} C_VEL
LIN {X 0,Y 126.673,Z 487.3,A -85,B 0,C 180,E1 -26328.261,E2 -26328.261} C_VEL
LIN {X 0,Y 124.196,Z 490.511,A -85,B 0,C 180,E1 -26330.463,E2 -26330.463} C_VEL
LIN {X 0,Y 118.038,Z 496.643,A -85,B 0,C 180,E1 -26335.557,E2 -26335.557} C_VEL
LIN {X 0,Y 113.688,Z 500.717,A -85,B 0,C 180,E1 -26340.363,E2 -26340.363} C_VEL
LIN {X 0,Y 109.356,Z 504.608,A -85,B 0,C 180,E1 -26347.322,E2 -26347.322} C_VEL
LIN {X 0,Y 107.902,Z 505.961,A -85,B 0,C 180,E1 -26350.997,E2 -26350.997} C_VEL
LIN {X 0,Y 106.469,Z 507.44,A -85,B 0,C 180,E1 -26358.581,E2 -26358.581} C_VEL
LIN {X 0,Y 106.527,Z 507.623,A -85,B 0,C 180,E1 -26362.421,E2 -26362.421} C_VEL
LIN {X 0,Y 106.908,Z 507.413,A -85,B 0,C 180,E1 -26366.233,E2 -26366.233} C_VEL
LIN {X 0,Y 107.409,Z 506.742,A -85,B 0,C 180,E1 -26370.003,E2 -26370.003} C_VEL
LIN {X 0,Y 106.839,Z 505.452,A -85,B 0,C 180,E1 -26373.774,E2 -26373.774} C_VEL
LIN {X 0,Y 106.51,Z 503.421,A -85,B 0,C 180,E1 -26378.208,E2 -26378.208} C_VEL
LIN {X 0,Y 106.702,Z 500.256,A -85,B 0,C 180,E1 -26383.331,E2 -26383.331} C_VEL
LIN {X 0,Y 107.877,Z 495.684,A -85,B 0,C 180,E1 -26389.013,E2 -26389.013} C_VEL
LIN {X 0,Y 110.086,Z 489.898,A -85,B 0,C 180,E1 -26394.52,E2 -26394.52} C_VEL
LIN {X 0,Y 113.479,Z 482.724,A -85,B 0,C 180,E1 -26399.703,E2 -26399.703} C_VEL
LIN {X 0,Y 116.293,Z 473.43,A -85,B 0,C 180,E1 -26405.041,E2 -26405.041} C_VEL
LIN {X 0,Y 118.914,Z 464.501,A -85,B 0,C 180,E1 -26409.116,E2 -26409.116} C_VEL
LIN {X 0,Y 121.236,Z 454.451,A -85,B 0,C 180,E1 -26412.936,E2 -26412.936} C_VEL
LIN {X 0,Y 122.968,Z 443.952,A -85,B 0,C 180,E1 -26416.324,E2 -26416.324} C_VEL
LIN {X 0,Y 123.877,Z 433.108,A -85,B 0,C 180,E1 -26419.432,E2 -26419.432} C_VEL
LIN {X 0,Y 123.897,Z 429.53,A -85,B 0,C 180,E1 -26420.424,E2 -26420.424} C_VEL
LIN {X 0,Y 120.735,Z 419.427,A -85,B 0,C 180,E1 -26424.586,E2 -26424.586} C_VEL
LIN {X 0,Y 118.004,Z 412.282,A -85,B 0,C 180,E1 -26427.84,E2 -26427.84} C_VEL
LIN {X 0,Y 115.942,Z 407.533,A -85,B 0,C 180,E1 -26430.245,E2 -26430.245} C_VEL
LIN {X 0,Y 113.115,Z 402.334,A -85,B 0,C 180,E1 -26433.477,E2 -26433.477} C_VEL
LIN {X 0,Y 112.302,Z 400.356,A -85,B 0,C 180,E1 -26434.534,E2 -26434.534} C_VEL
LIN {X 0,Y 109.267,Z 395.954,A -85,B 0,C 180,E1 -26438.295,E2 -26438.295} C_VEL
LIN {X 0,Y 108.107,Z 392.858,A -85,B 0,C 180,E1 -26440.292,E2 -26440.292} C_VEL
LIN {X 0,Y 107.986,Z 392.038,A -85,B 0,C 180,E1 -26442.483,E2 -26442.483} C_VEL
LIN {X 0,Y 108.312,Z 391.995,A -85,B 0,C 180,E1 -26448.776,E2 -26448.776} C_VEL
LIN {X 0,Y 108.468,Z 391.961,A -85,B 0,C 180,E1 -26456.286,E2 -26456.286} C_VEL
LIN {X 0,Y 108.953,Z 391.896,A -85,B 0,C 180,E1 -26460.001,E2 -26460.001} C_VEL
LIN {X 0,Y 108.344,Z 391.966,A -85,B 0,C 180,E1 -26467.455,E2 -26467.455} C_VEL
LIN {X 0,Y 108.209,Z 391.993,A -85,B 0,C 180,E1 -26473.025,E2 -26473.025} C_VEL
LIN {X 0,Y 107.904,Z 392.042,A -85,B 0,C 180,E1 -26479.131,E2 -26479.131} C_VEL
LIN {X 0,Y 107.601,Z 392.641,A -85,B 0,C 180,E1 -26482.267,E2 -26482.267} C_VEL
LIN {X 0,Y 107.137,Z 394.963,A -85,B 0,C 180,E1 -26486.317,E2 -26486.317} C_VEL
LIN {X 0,Y 107.142,Z 399.516,A -85,B 0,C 180,E1 -26491.133,E2 -26491.133} C_VEL
LIN {X 0,Y 108.215,Z 403.865,A -85,B 0,C 180,E1 -26494.723,E2 -26494.723} C_VEL
LIN {X 0,Y 112.761,Z 412.27,A -85,B 0,C 180,E1 -26501.951,E2 -26501.951} C_VEL
LIN {X 0,Y 115.772,Z 419.01,A -85,B 0,C 180,E1 -26506.76,E2 -26506.76} C_VEL
LIN {X 0,Y 118.333,Z 426.583,A -85,B 0,C 180,E1 -26511.547,E2 -26511.547} C_VEL
LIN {X 0,Y 119.974,Z 434.193,A -85,B 0,C 180,E1 -26516.025,E2 -26516.025} C_VEL
LIN {X 0,Y 120.547,Z 438.175,A -85,B 0,C 180,E1 -26518.349,E2 -26518.349} C_VEL
LIN {X 0,Y 120.526,Z 439.975,A -85,B 0,C 180,E1 -26519.319,E2 -26519.319} C_VEL
LIN {X 0,Y 116.372,Z 448.875,A -85,B 0,C 180,E1 -26523.065,E2 -26523.065} C_VEL
LIN {X 0,Y 111.865,Z 457.585,A -85,B 0,C 180,E1 -26527.852,E2 -26527.852} C_VEL
LIN {X 0,Y 108.091,Z 464.567,A -85,B 0,C 180,E1 -26532.984,E2 -26532.984} C_VEL
LIN {X 0,Y 105.125,Z 470.14,A -85,B 0,C 180,E1 -26538.427,E2 -26538.427} C_VEL
LIN {X 0,Y 102.85,Z 474.563,A -85,B 0,C 180,E1 -26544.114,E2 -26544.114} C_VEL
LIN {X 0,Y 101.321,Z 477.951,A -85,B 0,C 180,E1 -26549.997,E2 -26549.997} C_VEL
LIN {X 0,Y 101.017,Z 480.91,A -85,B 0,C 180,E1 -26557.995,E2 -26557.995} C_VEL
LIN {X 0,Y 101.906,Z 482.241,A -85,B 0,C 180,E1 -26565.086,E2 -26565.086} C_VEL
LIN {X 0,Y 103.181,Z 482.411,A -85,B 0,C 180,E1 -26569.908,E2 -26569.908} C_VEL
LIN {X 0,Y 106.603,Z 481.467,A -85,B 0,C 180,E1 -26577.48,E2 -26577.48} C_VEL
LIN {X 0,Y 108.887,Z 480.357,A -85,B 0,C 180,E1 -26581.085,E2 -26581.085} C_VEL
LIN {X 0,Y 112.878,Z 478.059,A -85,B 0,C 180,E1 -26585.961,E2 -26585.961} C_VEL
LIN {X 0,Y 117.895,Z 474.479,A -85,B 0,C 180,E1 -26590.972,E2 -26590.972} C_VEL
LIN {X 0,Y 123.393,Z 469.907,A -85,B 0,C 180,E1 -26595.39,E2 -26595.39} C_VEL
LIN {X 0,Y 130.578,Z 462.954,A -85,B 0,C 180,E1 -26600.079,E2 -26600.079} C_VEL
LIN {X 0,Y 132.779,Z 460.582,A -85,B 0,C 180,E1 -26601.323,E2 -26601.323} C_VEL
LIN {X 0,Y 133.335,Z 458.338,A -85,B 0,C 180,E1 -26603.38,E2 -26603.38} C_VEL
LIN {X 0,Y 133.823,Z 454.351,A -85,B 0,C 180,E1 -26607.165,E2 -26607.165} C_VEL
LIN {X 0,Y 133.938,Z 449.655,A -85,B 0,C 180,E1 -26611.819,E2 -26611.819} C_VEL
LIN {X 0,Y 133.634,Z 445.107,A -85,B 0,C 180,E1 -26616.768,E2 -26616.768} C_VEL
LIN {X 0,Y 133.36,Z 442.456,A -85,B 0,C 180,E1 -26619.967,E2 -26619.967} C_VEL
LIN {X 0,Y 132.888,Z 439.152,A -85,B 0,C 180,E1 -26624.666,E2 -26624.666} C_VEL
LIN {X 0,Y 132.658,Z 437.333,A -85,B 0,C 180,E1 -26627.765,E2 -26627.765} C_VEL
LIN {X 0,Y 132.402,Z 434.626,A -85,B 0,C 180,E1 -26633.905,E2 -26633.905} C_VEL
LIN {X 0,Y 132.679,Z 433.331,A -85,B 0,C 180,E1 -26636.963,E2 -26636.963} C_VEL
LIN {X 0,Y 132.918,Z 432.694,A -85,B 0,C 180,E1 -26639.999,E2 -26639.999} C_VEL
LIN {X 0,Y 132.749,Z 433.343,A -85,B 0,C 180,E1 -26643.034,E2 -26643.034} C_VEL
LIN {X 0,Y 132.746,Z 434.341,A -85,B 0,C 180,E1 -26646.078,E2 -26646.078} C_VEL
LIN {X 0,Y 132.886,Z 435.72,A -85,B 0,C 180,E1 -26649.129,E2 -26649.129} C_VEL
LIN {X 0,Y 133.277,Z 441.813,A -85,B 0,C 180,E1 -26656.859,E2 -26656.859} C_VEL
LIN {X 0,Y 133.826,Z 446.611,A -85,B 0,C 180,E1 -26661.568,E2 -26661.568} C_VEL
LIN {X 0,Y 134.337,Z 452.577,A -85,B 0,C 180,E1 -26666.404,E2 -26666.404} C_VEL
LIN {X 0,Y 134.538,Z 458.555,A -85,B 0,C 180,E1 -26670.618,E2 -26670.618} C_VEL
LIN {X 0,Y 134.364,Z 462.549,A -85,B 0,C 180,E1 -26673.191,E2 -26673.191} C_VEL
LIN {X 0,Y 130.385,Z 471.606,A -85,B 0,C 180,E1 -26677.344,E2 -26677.344} C_VEL
LIN {X 0,Y 126.07,Z 479.453,A -85,B 0,C 180,E1 -26681.431,E2 -26681.431} C_VEL
LIN {X 0,Y 121.283,Z 486.698,A -85,B 0,C 180,E1 -26685.947,E2 -26685.947} C_VEL
LIN {X 0,Y 117.777,Z 490.834,A -85,B 0,C 180,E1 -26688.978,E2 -26688.978} C_VEL
LIN {X 0,Y 112.219,Z 495.949,A -85,B 0,C 180,E1 -26693.493,E2 -26693.493} C_VEL
LIN {X 0,Y 107.514,Z 499.971,A -85,B 0,C 180,E1 -26698.473,E2 -26698.473} C_VEL
LIN {X 0,Y 102.808,Z 503.82,A -85,B 0,C 180,E1 -26705.788,E2 -26705.788} C_VEL
LIN {X 0,Y 101.156,Z 505.132,A -85,B 0,C 180,E1 -26709.676,E2 -26709.676} C_VEL
LIN {X 0,Y 99.464,Z 506.565,A -85,B 0,C 180,E1 -26717.765,E2 -26717.765} C_VEL
LIN {X 0,Y 99.457,Z 506.73,A -85,B 0,C 180,E1 -26721.878,E2 -26721.878} C_VEL
LIN {X 0,Y 99.819,Z 506.497,A -85,B 0,C 180,E1 -26725.966,E2 -26725.966} C_VEL
LIN {X 0,Y 100.32,Z 505.791,A -85,B 0,C 180,E1 -26730.003,E2 -26730.003} C_VEL
LIN {X 0,Y 99.719,Z 504.474,A -85,B 0,C 180,E1 -26734.044,E2 -26734.044} C_VEL
LIN {X 0,Y 99.44,Z 501.664,A -85,B 0,C 180,E1 -26740.178,E2 -26740.178} C_VEL
LIN {X 0,Y 100.073,Z 497.783,A -85,B 0,C 180,E1 -26746.318,E2 -26746.318} C_VEL
LIN {X 0,Y 101.801,Z 492.761,A -85,B 0,C 180,E1 -26752.318,E2 -26752.318} C_VEL
LIN {X 0,Y 104.766,Z 486.483,A -85,B 0,C 180,E1 -26758.01,E2 -26758.01} C_VEL
LIN {X 0,Y 107.141,Z 481.446,A -85,B 0,C 180,E1 -26761.656,E2 -26761.656} C_VEL
LIN {X 0,Y 110.278,Z 472.062,A -85,B 0,C 180,E1 -26767.263,E2 -26767.263} C_VEL
LIN {X 0,Y 113.103,Z 463.193,A -85,B 0,C 180,E1 -26771.452,E2 -26771.452} C_VEL
LIN {X 0,Y 115.7,Z 452.8,A -85,B 0,C 180,E1 -26775.543,E2 -26775.543} C_VEL
LIN {X 0,Y 117.619,Z 441.691,A -85,B 0,C 180,E1 -26779.25,E2 -26779.25} C_VEL
LIN {X 0,Y 118.436,Z 433.181,A -85,B 0,C 180,E1 -26781.838,E2 -26781.838} C_VEL
LIN {X 0,Y 116.982,Z 427.026,A -85,B 0,C 180,E1 -26784.52,E2 -26784.52} C_VEL
LIN {X 0,Y 114.364,Z 418.709,A -85,B 0,C 180,E1 -26788.511,E2 -26788.511} C_VEL
LIN {X 0,Y 111.644,Z 411.917,A -85,B 0,C 180,E1 -26792.326,E2 -26792.326} C_VEL
LIN {X 0,Y 109.486,Z 407.033,A -85,B 0,C 180,E1 -26795.467,E2 -26795.467} C_VEL
LIN {X 0,Y 108.717,Z 405.585,A -85,B 0,C 180,E1 -26796.549,E2 -26796.549} C_VEL
LIN {X 0,Y 106.347,Z 401.303,A -85,B 0,C 180,E1 -26800.204,E2 -26800.204} C_VEL
LIN {X 0,Y 105.517,Z 398.981,A -85,B 0,C 180,E1 -26801.808,E2 -26801.808} C_VEL
LIN {X 0,Y 102.55,Z 396.318,A -85,B 0,C 180,E1 -26806.845,E2 -26806.845} C_VEL
LIN {X 0,Y 101.28,Z 393.195,A -85,B 0,C 180,E1 -26810.389,E2 -26810.389} C_VEL
LIN {X 0,Y 101.258,Z 392.873,A -85,B 0,C 180,E1 -26811.016,E2 -26811.016} C_VEL
LIN {X 0,Y 101.877,Z 392.776,A -85,B 0,C 180,E1 -26820.001,E2 -26820.001} C_VEL
LIN {X 0,Y 101.284,Z 392.847,A -85,B 0,C 180,E1 -26827.978,E2 -26827.978} C_VEL
LIN {X 0,Y 101.12,Z 392.873,A -85,B 0,C 180,E1 -26833.326,E2 -26833.326} C_VEL
LIN {X 0,Y 100.88,Z 393.082,A -85,B 0,C 180,E1 -26839.59,E2 -26839.59} C_VEL
LIN {X 0,Y 101.543,Z 395.214,A -85,B 0,C 180,E1 -26842.108,E2 -26842.108} C_VEL
LIN {X 0,Y 103.625,Z 397.819,A -85,B 0,C 180,E1 -26846.782,E2 -26846.782} C_VEL
LIN {X 0,Y 105.004,Z 398.721,A -85,B 0,C 180,E1 -26849.063,E2 -26849.063} C_VEL
LIN {X 0,Y 105.776,Z 400.86,A -85,B 0,C 180,E1 -26850.857,E2 -26850.857} C_VEL
LIN {X 0,Y 108.215,Z 403.865,A -85,B 0,C 180,E1 -26854.723,E2 -26854.723} C_VEL
LIN {X 0,Y 109.237,Z 407.511,A -85,B 0,C 180,E1 -26857.132,E2 -26857.132} C_VEL
LIN {X 0,Y 110.082,Z 414.471,A -85,B 0,C 180,E1 -26860.808,E2 -26860.808} C_VEL
LIN {X 0,Y 110.814,Z 422.812,A -85,B 0,C 180,E1 -26865.27,E2 -26865.27} C_VEL
LIN {X 0,Y 111.367,Z 425.261,A -85,B 0,C 180,E1 -26866.872,E2 -26866.872} C_VEL
LIN {X 0,Y 113.23,Z 432.284,A -85,B 0,C 180,E1 -26871.631,E2 -26871.631} C_VEL
LIN {X 0,Y 114.346,Z 439.742,A -85,B 0,C 180,E1 -26876.413,E2 -26876.413} C_VEL
LIN {X 0,Y 114.443,Z 441.44,A -85,B 0,C 180,E1 -26877.494,E2 -26877.494} C_VEL
LIN {X 0,Y 110.156,Z 450.22,A -85,B 0,C 180,E1 -26881.409,E2 -26881.409} C_VEL
LIN {X 0,Y 105.386,Z 458.847,A -85,B 0,C 180,E1 -26886.411,E2 -26886.411} C_VEL
LIN {X 0,Y 101.388,Z 465.731,A -85,B 0,C 180,E1 -26891.821,E2 -26891.821} C_VEL
LIN {X 0,Y 98.239,Z 471.247,A -85,B 0,C 180,E1 -26897.604,E2 -26897.604} C_VEL
LIN {X 0,Y 95.826,Z 475.618,A -85,B 0,C 180,E1 -26903.681,E2 -26903.681} C_VEL
LIN {X 0,Y 94.244,Z 478.957,A -85,B 0,C 180,E1 -26909.997,E2 -26909.997} C_VEL
LIN {X 0,Y 93.993,Z 481.871,A -85,B 0,C 180,E1 -26918.597,E2 -26918.597} C_VEL
LIN {X 0,Y 94.975,Z 483.111,A -85,B 0,C 180,E1 -26925.845,E2 -26925.845} C_VEL
LIN {X 0,Y 96.504,Z 483.281,A -85,B 0,C 180,E1 -26931.351,E2 -26931.351} C_VEL
LIN {X 0,Y 98.207,Z 482.979,A -85,B 0,C 180,E1 -26935.425,E2 -26935.425} C_VEL
LIN {X 0,Y 100.326,Z 482.271,A -85,B 0,C 180,E1 -26939.361,E2 -26939.361} C_VEL
LIN {X 0,Y 102.844,Z 481.131,A -85,B 0,C 180,E1 -26943.137,E2 -26943.137} C_VEL
LIN {X 0,Y 106.855,Z 478.982,A -85,B 0,C 180,E1 -26947.882,E2 -26947.882} C_VEL
LIN {X 0,Y 112.599,Z 475.151,A -85,B 0,C 180,E1 -26953.356,E2 -26953.356} C_VEL
LIN {X 0,Y 118.475,Z 470.521,A -85,B 0,C 180,E1 -26957.856,E2 -26957.856} C_VEL
LIN {X 0,Y 124.983,Z 464.604,A -85,B 0,C 180,E1 -26961.925,E2 -26961.925} C_VEL
LIN {X 0,Y 127.075,Z 462.338,A -85,B 0,C 180,E1 -26963.311,E2 -26963.311} C_VEL
LIN {X 0,Y 127.761,Z 459.21,A -85,B 0,C 180,E1 -26966.626,E2 -26966.626} C_VEL
LIN {X 0,Y 128.319,Z 455.012,A -85,B 0,C 180,E1 -26971.196,E2 -26971.196} C_VEL
LIN {X 0,Y 128.529,Z 451.028,A -85,B 0,C 180,E1 -26975.788,E2 -26975.788} C_VEL
LIN {X 0,Y 128.435,Z 447.222,A -85,B 0,C 180,E1 -26980.832,E2 -26980.832} C_VEL
LIN {X 0,Y 128.326,Z 445.136,A -85,B 0,C 180,E1 -26984.107,E2 -26984.107} C_VEL
LIN {X 0,Y 128.257,Z 443.294,A -85,B 0,C 180,E1 -26987.338,E2 -26987.338} C_VEL
LIN {X 0,Y 128.231,Z 441.782,A -85,B 0,C 180,E1 -26990.572,E2 -26990.572} C_VEL
LIN {X 0,Y 128.707,Z 439.402,A -85,B 0,C 180,E1 -26996.869,E2 -26996.869} C_VEL
LIN {X 0,Y 129.076,Z 438.706,A -85,B 0,C 180,E1 -26999.999,E2 -26999.999} C_VEL
LIN {X 0,Y 128.891,Z 439.409,A -85,B 0,C 180,E1 -27003.125,E2 -27003.125} C_VEL
LIN {X 0,Y 128.852,Z 440.476,A -85,B 0,C 180,E1 -27006.262,E2 -27006.262} C_VEL
LIN {X 0,Y 128.811,Z 442.121,A -85,B 0,C 180,E1 -27009.42,E2 -27009.42} C_VEL
LIN {X 0,Y 128.862,Z 446.867,A -85,B 0,C 180,E1 -27015.824,E2 -27015.824} C_VEL
LIN {X 0,Y 129.096,Z 451.525,A -85,B 0,C 180,E1 -27020.725,E2 -27020.725} C_VEL
LIN {X 0,Y 129.201,Z 456.273,A -85,B 0,C 180,E1 -27024.933,E2 -27024.933} C_VEL
LIN {X 0,Y 129.031,Z 462.035,A -85,B 0,C 180,E1 -27029.374,E2 -27029.374} C_VEL
LIN {X 0,Y 128.842,Z 464.547,A -85,B 0,C 180,E1 -27031.209,E2 -27031.209} C_VEL
LIN {X 0,Y 128.45,Z 465.914,A -85,B 0,C 180,E1 -27032.003,E2 -27032.003} C_VEL
LIN {X 0,Y 124.048,Z 474.257,A -85,B 0,C 180,E1 -27036.167,E2 -27036.167} C_VEL
LIN {X 0,Y 118.919,Z 482.203,A -85,B 0,C 180,E1 -27040.763,E2 -27040.763} C_VEL
LIN {X 0,Y 114.294,Z 488.208,A -85,B 0,C 180,E1 -27045.001,E2 -27045.001} C_VEL
LIN {X 0,Y 110.429,Z 492.03,A -85,B 0,C 180,E1 -27048.072,E2 -27048.072} C_VEL
LIN {X 0,Y 104.794,Z 496.719,A -85,B 0,C 180,E1 -27052.877,E2 -27052.877} C_VEL
LIN {X 0,Y 100.049,Z 500.359,A -85,B 0,C 180,E1 -27058.211,E2 -27058.211} C_VEL
LIN {X 0,Y 96.318,Z 503.03,A -85,B 0,C 180,E1 -27064.04,E2 -27064.04} C_VEL
LIN {X 0,Y 93.213,Z 505.182,A -85,B 0,C 180,E1 -27072.45,E2 -27072.45} C_VEL
LIN {X 0,Y 92.403,Z 505.838,A -85,B 0,C 180,E1 -27081.396,E2 -27081.396} C_VEL
LIN {X 0,Y 92.732,Z 505.571,A -85,B 0,C 180,E1 -27085.657,E2 -27085.657} C_VEL
LIN {X 0,Y 93.213,Z 504.838,A -85,B 0,C 180,E1 -27090.003,E2 -27090.003} C_VEL
LIN {X 0,Y 92.602,Z 503.496,A -85,B 0,C 180,E1 -27094.356,E2 -27094.356} C_VEL
LIN {X 0,Y 92.384,Z 500.634,A -85,B 0,C 180,E1 -27100.967,E2 -27100.967} C_VEL
LIN {X 0,Y 93.211,Z 496.707,A -85,B 0,C 180,E1 -27107.557,E2 -27107.557} C_VEL
LIN {X 0,Y 95.192,Z 491.631,A -85,B 0,C 180,E1 -27113.961,E2 -27113.961} C_VEL
LIN {X 0,Y 98.527,Z 485.305,A -85,B 0,C 180,E1 -27119.958,E2 -27119.958} C_VEL
LIN {X 0,Y 100.879,Z 480.147,A -85,B 0,C 180,E1 -27123.876,E2 -27123.876} C_VEL
LIN {X 0,Y 104.428,Z 470.677,A -85,B 0,C 180,E1 -27129.747,E2 -27129.747} C_VEL
LIN {X 0,Y 107.323,Z 462.191,A -85,B 0,C 180,E1 -27133.919,E2 -27133.919} C_VEL
LIN {X 0,Y 110.382,Z 451.083,A -85,B 0,C 180,E1 -27138.432,E2 -27138.432} C_VEL
LIN {X 0,Y 112.427,Z 439.865,A -85,B 0,C 180,E1 -27142.354,E2 -27142.354} C_VEL
LIN {X 0,Y 112.928,Z 435.62,A -85,B 0,C 180,E1 -27143.755,E2 -27143.755} C_VEL
LIN {X 0,Y 110.773,Z 426.264,A -85,B 0,C 180,E1 -27148.439,E2 -27148.439} C_VEL
LIN {X 0,Y 107.741,Z 417.069,A -85,B 0,C 180,E1 -27153.877,E2 -27153.877} C_VEL
LIN {X 0,Y 105.462,Z 411.323,A -85,B 0,C 180,E1 -27157.986,E2 -27157.986} C_VEL
LIN {X 0,Y 103.337,Z 406.866,A -85,B 0,C 180,E1 -27161.983,E2 -27161.983} C_VEL
LIN {X 0,Y 102.83,Z 405.147,A -85,B 0,C 180,E1 -27163.295,E2 -27163.295} C_VEL
LIN {X 0,Y 100.534,Z 403.02,A -85,B 0,C 180,E1 -27167.639,E2 -27167.639} C_VEL
LIN {X 0,Y 99.269,Z 399.667,A -85,B 0,C 180,E1 -27171.861,E2 -27171.861} C_VEL
LIN {X 0,Y 97.231,Z 398.17,A -85,B 0,C 180,E1 -27180.001,E2 -27180.001} C_VEL
LIN {X 0,Y 97.112,Z 398.662,A -85,B 0,C 180,E1 -27191.48,E2 -27191.48} C_VEL
LIN {X 0,Y 98.708,Z 399.823,A -85,B 0,C 180,E1 -27198.554,E2 -27198.554} C_VEL
LIN {X 0,Y 99.127,Z 401.497,A -85,B 0,C 180,E1 -27200.764,E2 -27200.764} C_VEL
LIN {X 0,Y 100.476,Z 403.77,A -85,B 0,C 180,E1 -27204.816,E2 -27204.816} C_VEL
LIN {X 0,Y 101.396,Z 404.583,A -85,B 0,C 180,E1 -27206.779,E2 -27206.779} C_VEL
LIN {X 0,Y 102.284,Z 405.891,A -85,B 0,C 180,E1 -27208.75,E2 -27208.75} C_VEL
LIN {X 0,Y 105.109,Z 410.906,A -85,B 0,C 180,E1 -27214.636,E2 -27214.636} C_VEL
LIN {X 0,Y 108.193,Z 417.064,A -85,B 0,C 180,E1 -27220.511,E2 -27220.511} C_VEL
LIN {X 0,Y 110.896,Z 423.791,A -85,B 0,C 180,E1 -27225.8,E2 -27225.8} C_VEL
LIN {X 0,Y 111.367,Z 425.261,A -85,B 0,C 180,E1 -27226.872,E2 -27226.872} C_VEL
LIN {X 0,Y 111.523,Z 428.009,A -85,B 0,C 180,E1 -27228.358,E2 -27228.358} C_VEL
LIN {X 0,Y 110.119,Z 433.308,A -85,B 0,C 180,E1 -27230.418,E2 -27230.418} C_VEL
LIN {X 0,Y 108.457,Z 438.463,A -85,B 0,C 180,E1 -27232.547,E2 -27232.547} C_VEL
LIN {X 0,Y 108.217,Z 441.118,A -85,B 0,C 180,E1 -27234.115,E2 -27234.115} C_VEL
LIN {X 0,Y 108.329,Z 442.945,A -85,B 0,C 180,E1 -27235.409,E2 -27235.409} C_VEL
LIN {X 0,Y 107.753,Z 444.768,A -85,B 0,C 180,E1 -27236.328,E2 -27236.328} C_VEL
LIN {X 0,Y 103.167,Z 453.132,A -85,B 0,C 180,E1 -27240.4,E2 -27240.4} C_VEL
LIN {X 0,Y 98.226,Z 461.304,A -85,B 0,C 180,E1 -27245.704,E2 -27245.704} C_VEL
LIN {X 0,Y 94.732,Z 466.895,A -85,B 0,C 180,E1 -27250.494,E2 -27250.494} C_VEL
LIN {X 0,Y 91.376,Z 472.353,A -85,B 0,C 180,E1 -27256.656,E2 -27256.656} C_VEL
LIN {X 0,Y 88.807,Z 476.674,A -85,B 0,C 180,E1 -27263.179,E2 -27263.179} C_VEL
LIN {X 0,Y 87.167,Z 479.964,A -85,B 0,C 180,E1 -27269.997,E2 -27269.997} C_VEL
LIN {X 0,Y 86.982,Z 482.831,A -85,B 0,C 180,E1 -27279.296,E2 -27279.296} C_VEL
LIN {X 0,Y 88.051,Z 483.979,A -85,B 0,C 180,E1 -27286.698,E2 -27286.698} C_VEL
LIN {X 0,Y 89.914,Z 484.148,A -85,B 0,C 180,E1 -27293.002,E2 -27293.002} C_VEL
LIN {X 0,Y 91.807,Z 483.826,A -85,B 0,C 180,E1 -27297.339,E2 -27297.339} C_VEL
LIN {X 0,Y 94.179,Z 483.069,A -85,B 0,C 180,E1 -27301.488,E2 -27301.488} C_VEL
LIN {X 0,Y 96.951,Z 481.905,A -85,B 0,C 180,E1 -27305.441,E2 -27305.441} C_VEL
LIN {X 0,Y 100.978,Z 479.898,A -85,B 0,C 180,E1 -27310.038,E2 -27310.038} C_VEL
LIN {X 0,Y 107.507,Z 475.823,A -85,B 0,C 180,E1 -27315.976,E2 -27315.976} C_VEL
LIN {X 0,Y 113.803,Z 471.135,A -85,B 0,C 180,E1 -27320.525,E2 -27320.525} C_VEL
LIN {X 0,Y 120.703,Z 465.155,A -85,B 0,C 180,E1 -27324.598,E2 -27324.598} C_VEL
LIN {X 0,Y 121.617,Z 463.107,A -85,B 0,C 180,E1 -27326.802,E2 -27326.802} C_VEL
LIN {X 0,Y 122.463,Z 459.579,A -85,B 0,C 180,E1 -27331.058,E2 -27331.058} C_VEL
LIN {X 0,Y 123.108,Z 455.375,A -85,B 0,C 180,E1 -27336.445,E2 -27336.445} C_VEL
LIN {X 0,Y 123.361,Z 451.818,A -85,B 0,C 180,E1 -27341.738,E2 -27341.738} C_VEL
LIN {X 0,Y 123.502,Z 449.03,A -85,B 0,C 180,E1 -27346.842,E2 -27346.842} C_VEL
LIN {X 0,Y 123.681,Z 447.538,A -85,B 0,C 180,E1 -27350.184,E2 -27350.184} C_VEL
LIN {X 0,Y 124.39,Z 445.234,A -85,B 0,C 180,E1 -27356.76,E2 -27356.76} C_VEL
LIN {X 0,Y 124.905,Z 444.519,A -85,B 0,C 180,E1 -27359.999,E2 -27359.999} C_VEL
LIN {X 0,Y 124.713,Z 445.257,A -85,B 0,C 180,E1 -27363.23,E2 -27363.23} C_VEL
LIN {X 0,Y 124.584,Z 446.454,A -85,B 0,C 180,E1 -27366.477,E2 -27366.477} C_VEL
LIN {X 0,Y 124.273,Z 449.154,A -85,B 0,C 180,E1 -27371.046,E2 -27371.046} C_VEL
LIN {X 0,Y 124.166,Z 452.612,A -85,B 0,C 180,E1 -27375.806,E2 -27375.806} C_VEL
LIN {X 0,Y 124.075,Z 457.349,A -85,B 0,C 180,E1 -27381.023,E2 -27381.023} C_VEL
LIN {X 0,Y 123.832,Z 461.416,A -85,B 0,C 180,E1 -27384.766,E2 -27384.766} C_VEL
LIN {X 0,Y 123.194,Z 467.142,A -85,B 0,C 180,E1 -27389.506,E2 -27389.506} C_VEL
LIN {X 0,Y 122.494,Z 468.928,A -85,B 0,C 180,E1 -27390.619,E2 -27390.619} C_VEL
LIN {X 0,Y 117.734,Z 476.641,A -85,B 0,C 180,E1 -27394.84,E2 -27394.84} C_VEL
LIN {X 0,Y 112.48,Z 483.701,A -85,B 0,C 180,E1 -27399.346,E2 -27399.346} C_VEL
LIN {X 0,Y 109.216,Z 487.577,A -85,B 0,C 180,E1 -27402.271,E2 -27402.271} C_VEL
LIN {X 0,Y 105.203,Z 491.36,A -85,B 0,C 180,E1 -27405.461,E2 -27405.461} C_VEL
LIN {X 0,Y 99.189,Z 496.001,A -85,B 0,C 180,E1 -27410.384,E2 -27410.384} C_VEL
LIN {X 0,Y 94.036,Z 499.594,A -85,B 0,C 180,E1 -27415.911,E2 -27415.911} C_VEL
LIN {X 0,Y 89.94,Z 502.233,A -85,B 0,C 180,E1 -27422.044,E2 -27422.044} C_VEL
LIN {X 0,Y 86.425,Z 504.33,A -85,B 0,C 180,E1 -27431.021,E2 -27431.021} C_VEL
LIN {X 0,Y 85.327,Z 504.938,A -85,B 0,C 180,E1 -27440.522,E2 -27440.522} C_VEL
LIN {X 0,Y 85.648,Z 504.638,A -85,B 0,C 180,E1 -27445.297,E2 -27445.297} C_VEL
LIN {X 0,Y 86.106,Z 503.884,A -85,B 0,C 180,E1 -27450.003,E2 -27450.003} C_VEL
LIN {X 0,Y 85.314,Z 501.036,A -85,B 0,C 180,E1 -27458.689,E2 -27458.689} C_VEL
LIN {X 0,Y 85.906,Z 497.098,A -85,B 0,C 180,E1 -27466.642,E2 -27466.642} C_VEL
LIN {X 0,Y 87.753,Z 492.363,A -85,B 0,C 180,E1 -27473.609,E2 -27473.609} C_VEL
LIN {X 0,Y 91.678,Z 485.259,A -85,B 0,C 180,E1 -27481.165,E2 -27481.165} C_VEL
LIN {X 0,Y 94.172,Z 480.436,A -85,B 0,C 180,E1 -27485.191,E2 -27485.191} C_VEL
LIN {X 0,Y 98.085,Z 471.02,A -85,B 0,C 180,E1 -27491.517,E2 -27491.517} C_VEL
LIN {X 0,Y 101.548,Z 461.842,A -85,B 0,C 180,E1 -27496.343,E2 -27496.343} C_VEL
LIN {X 0,Y 104.621,Z 452.033,A -85,B 0,C 180,E1 -27500.585,E2 -27500.585} C_VEL
LIN {X 0,Y 107.007,Z 441.393,A -85,B 0,C 180,E1 -27504.603,E2 -27504.603} C_VEL
LIN {X 0,Y 107.445,Z 438.446,A -85,B 0,C 180,E1 -27505.657,E2 -27505.657} C_VEL
LIN {X 0,Y 105.702,Z 429.391,A -85,B 0,C 180,E1 -27510.748,E2 -27510.748} C_VEL
LIN {X 0,Y 103.918,Z 422.779,A -85,B 0,C 180,E1 -27514.996,E2 -27514.996} C_VEL
LIN {X 0,Y 102.277,Z 417.589,A -85,B 0,C 180,E1 -27518.854,E2 -27518.854} C_VEL
LIN {X 0,Y 100.192,Z 412.452,A -85,B 0,C 180,E1 -27523.706,E2 -27523.706} C_VEL
LIN {X 0,Y 99.358,Z 411.01,A -85,B 0,C 180,E1 -27525.667,E2 -27525.667} C_VEL
LIN {X 0,Y 97.635,Z 408.449,A -85,B 0,C 180,E1 -27530.157,E2 -27530.157} C_VEL
LIN {X 0,Y 97.111,Z 406.4,A -85,B 0,C 180,E1 -27532.725,E2 -27532.725} C_VEL
LIN {X 0,Y 95.419,Z 405.059,A -85,B 0,C 180,E1 -27540.001,E2 -27540.001} C_VEL
LIN {X 0,Y 94.928,Z 405.228,A -85,B 0,C 180,E1 -27548.516,E2 -27548.516} C_VEL
LIN {X 0,Y 96.158,Z 406.254,A -85,B 0,C 180,E1 -27557,E2 -27557} C_VEL
LIN {X 0,Y 96.902,Z 408.719,A -85,B 0,C 180,E1 -27561.263,E2 -27561.263} C_VEL
LIN {X 0,Y 99,Z 411.81,A -85,B 0,C 180,E1 -27567.481,E2 -27567.481} C_VEL
LIN {X 0,Y 101.364,Z 416.693,A -85,B 0,C 180,E1 -27573.689,E2 -27573.689} C_VEL
LIN {X 0,Y 103.638,Z 421.972,A -85,B 0,C 180,E1 -27579.157,E2 -27579.157} C_VEL
LIN {X 0,Y 105.691,Z 427.834,A -85,B 0,C 180,E1 -27584.282,E2 -27584.282} C_VEL
LIN {X 0,Y 107.246,Z 434.009,A -85,B 0,C 180,E1 -27589.053,E2 -27589.053} C_VEL
LIN {X 0,Y 108.217,Z 441.118,A -85,B 0,C 180,E1 -27594.115,E2 -27594.115} C_VEL
LIN {X 0,Y 107.676,Z 443.292,A -85,B 0,C 180,E1 -27595.269,E2 -27595.269} C_VEL
LIN {X 0,Y 106.106,Z 445.67,A -85,B 0,C 180,E1 -27596.098,E2 -27596.098} C_VEL
LIN {X 0,Y 103.528,Z 448.461,A -85,B 0,C 180,E1 -27596.803,E2 -27596.803} C_VEL
LIN {X 0,Y 98.483,Z 453.25,A -85,B 0,C 180,E1 -27598.018,E2 -27598.018} C_VEL
LIN {X 0,Y 96.136,Z 456.019,A -85,B 0,C 180,E1 -27599.316,E2 -27599.316} C_VEL
LIN {X 0,Y 91.059,Z 463.752,A -85,B 0,C 180,E1 -27604.878,E2 -27604.878} C_VEL
LIN {X 0,Y 86.858,Z 470.012,A -85,B 0,C 180,E1 -27611.112,E2 -27611.112} C_VEL
LIN {X 0,Y 83.472,Z 475.024,A -85,B 0,C 180,E1 -27617.845,E2 -27617.845} C_VEL
LIN {X 0,Y 81.092,Z 478.936,A -85,B 0,C 180,E1 -27625.024,E2 -27625.024} C_VEL
LIN {X 0,Y 80.091,Z 480.97,A -85,B 0,C 180,E1 -27629.996,E2 -27629.996} C_VEL
LIN {X 0,Y 79.788,Z 482.573,A -85,B 0,C 180,E1 -27635.05,E2 -27635.05} C_VEL
LIN {X 0,Y 79.987,Z 483.783,A -85,B 0,C 180,E1 -27640.117,E2 -27640.117} C_VEL
LIN {X 0,Y 81.747,Z 484.984,A -85,B 0,C 180,E1 -27650.11,E2 -27650.11} C_VEL
LIN {X 0,Y 85.536,Z 484.662,A -85,B 0,C 180,E1 -27659.533,E2 -27659.533} C_VEL
LIN {X 0,Y 91.237,Z 482.678,A -85,B 0,C 180,E1 -27668.038,E2 -27668.038} C_VEL
LIN {X 0,Y 95.32,Z 480.787,A -85,B 0,C 180,E1 -27672.496,E2 -27672.496} C_VEL
LIN {X 0,Y 102.651,Z 476.497,A -85,B 0,C 180,E1 -27678.856,E2 -27678.856} C_VEL
LIN {X 0,Y 109.402,Z 471.749,A -85,B 0,C 180,E1 -27683.413,E2 -27683.413} C_VEL
LIN {X 0,Y 115.136,Z 467.074,A -85,B 0,C 180,E1 -27686.675,E2 -27686.675} C_VEL
LIN {X 0,Y 116.415,Z 463.736,A -85,B 0,C 180,E1 -27691.12,E2 -27691.12} C_VEL
LIN {X 0,Y 117.229,Z 460.848,A -85,B 0,C 180,E1 -27695.186,E2 -27695.186} C_VEL
LIN {X 0,Y 117.743,Z 458.378,A -85,B 0,C 180,E1 -27699.013,E2 -27699.013} C_VEL
LIN {X 0,Y 118.144,Z 456.236,A -85,B 0,C 180,E1 -27702.696,E2 -27702.696} C_VEL
LIN {X 0,Y 118.447,Z 454.491,A -85,B 0,C 180,E1 -27706.27,E2 -27706.27} C_VEL
LIN {X 0,Y 118.747,Z 453.018,A -85,B 0,C 180,E1 -27709.772,E2 -27709.772} C_VEL
LIN {X 0,Y 119.721,Z 450.804,A -85,B 0,C 180,E1 -27716.634,E2 -27716.634} C_VEL
LIN {X 0,Y 120.411,Z 450.108,A -85,B 0,C 180,E1 -27719.999,E2 -27719.999} C_VEL
LIN {X 0,Y 120.194,Z 450.903,A -85,B 0,C 180,E1 -27723.351,E2 -27723.351} C_VEL
LIN {X 0,Y 119.951,Z 452.214,A -85,B 0,C 180,E1 -27726.729,E2 -27726.729} C_VEL
LIN {X 0,Y 119.423,Z 455.238,A -85,B 0,C 180,E1 -27731.886,E2 -27731.886} C_VEL
LIN {X 0,Y 119.177,Z 457.802,A -85,B 0,C 180,E1 -27735.451,E2 -27735.451} C_VEL
LIN {X 0,Y 118.928,Z 460.702,A -85,B 0,C 180,E1 -27739.009,E2 -27739.009} C_VEL
LIN {X 0,Y 118.511,Z 464.218,A -85,B 0,C 180,E1 -27742.672,E2 -27742.672} C_VEL
LIN {X 0,Y 117.577,Z 469.496,A -85,B 0,C 180,E1 -27747.556,E2 -27747.556} C_VEL
LIN {X 0,Y 116.941,Z 471.069,A -85,B 0,C 180,E1 -27748.736,E2 -27748.736} C_VEL
LIN {X 0,Y 112.47,Z 477.474,A -85,B 0,C 180,E1 -27752.484,E2 -27752.484} C_VEL
LIN {X 0,Y 106.335,Z 484.792,A -85,B 0,C 180,E1 -27757.527,E2 -27757.527} C_VEL
LIN {X 0,Y 102.342,Z 488.88,A -85,B 0,C 180,E1 -27760.945,E2 -27760.945} C_VEL
LIN {X 0,Y 97.999,Z 492.369,A -85,B 0,C 180,E1 -27764.185,E2 -27764.185} C_VEL
LIN {X 0,Y 91.824,Z 496.595,A -85,B 0,C 180,E1 -27769.419,E2 -27769.419} C_VEL
LIN {X 0,Y 86.571,Z 499.801,A -85,B 0,C 180,E1 -27775.374,E2 -27775.374} C_VEL
LIN {X 0,Y 83.694,Z 501.427,A -85,B 0,C 180,E1 -27779.75,E2 -27779.75} C_VEL
LIN {X 0,Y 79.709,Z 503.478,A -85,B 0,C 180,E1 -27789.352,E2 -27789.352} C_VEL
LIN {X 0,Y 78.286,Z 504.034,A -85,B 0,C 180,E1 -27799.66,E2 -27799.66} C_VEL
LIN {X 0,Y 78.566,Z 503.705,A -85,B 0,C 180,E1 -27804.872,E2 -27804.872} C_VEL
LIN {X 0,Y 78.999,Z 502.929,A -85,B 0,C 180,E1 -27810.004,E2 -27810.004} C_VEL
LIN {X 0,Y 78.238,Z 500.258,A -85,B 0,C 180,E1 -27818.85,E2 -27818.85} C_VEL
LIN {X 0,Y 79.065,Z 496.033,A -85,B 0,C 180,E1 -27828.13,E2 -27828.13} C_VEL
LIN {X 0,Y 81.222,Z 491.239,A -85,B 0,C 180,E1 -27835.639,E2 -27835.639} C_VEL
LIN {X 0,Y 84.877,Z 485.214,A -85,B 0,C 180,E1 -27842.566,E2 -27842.566} C_VEL
LIN {X 0,Y 87.387,Z 480.917,A -85,B 0,C 180,E1 -27846.465,E2 -27846.465} C_VEL
LIN {X 0,Y 91.083,Z 472.992,A -85,B 0,C 180,E1 -27852.471,E2 -27852.471} C_VEL
LIN {X 0,Y 94.971,Z 464.087,A -85,B 0,C 180,E1 -27857.738,E2 -27857.738} C_VEL
LIN {X 0,Y 98.618,Z 454.233,A -85,B 0,C 180,E1 -27862.425,E2 -27862.425} C_VEL
LIN {X 0,Y 101.587,Z 443.381,A -85,B 0,C 180,E1 -27866.864,E2 -27866.864} C_VEL
LIN {X 0,Y 101.927,Z 440.927,A -85,B 0,C 180,E1 -27867.941,E2 -27867.941} C_VEL
LIN {X 0,Y 100.76,Z 432.707,A -85,B 0,C 180,E1 -27873.04,E2 -27873.04} C_VEL
LIN {X 0,Y 99.475,Z 427.094,A -85,B 0,C 180,E1 -27877.133,E2 -27877.133} C_VEL
LIN {X 0,Y 98.19,Z 422.193,A -85,B 0,C 180,E1 -27881.211,E2 -27881.211} C_VEL
LIN {X 0,Y 96.881,Z 418.188,A -85,B 0,C 180,E1 -27885.293,E2 -27885.293} C_VEL
LIN {X 0,Y 94.91,Z 414.591,A -85,B 0,C 180,E1 -27891.484,E2 -27891.484} C_VEL
LIN {X 0,Y 93.993,Z 412.694,A -85,B 0,C 180,E1 -27895.713,E2 -27895.713} C_VEL
LIN {X 0,Y 93.233,Z 411.847,A -85,B 0,C 180,E1 -27900.001,E2 -27900.001} C_VEL
LIN {X 0,Y 92.669,Z 412.059,A -85,B 0,C 180,E1 -27909.608,E2 -27909.608} C_VEL
LIN {X 0,Y 92.984,Z 412.394,A -85,B 0,C 180,E1 -27913.107,E2 -27913.107} C_VEL
LIN {X 0,Y 93.634,Z 413.421,A -85,B 0,C 180,E1 -27917.473,E2 -27917.473} C_VEL
LIN {X 0,Y 95.519,Z 417.672,A -85,B 0,C 180,E1 -27926.198,E2 -27926.198} C_VEL
LIN {X 0,Y 97.229,Z 421.822,A -85,B 0,C 180,E1 -27932.076,E2 -27932.076} C_VEL
LIN {X 0,Y 99.419,Z 427.927,A -85,B 0,C 180,E1 -27938.954,E2 -27938.954} C_VEL
LIN {X 0,Y 100.925,Z 433.48,A -85,B 0,C 180,E1 -27944.137,E2 -27944.137} C_VEL
LIN {X 0,Y 101.827,Z 438.687,A -85,B 0,C 180,E1 -27948.482,E2 -27948.482} C_VEL
LIN {X 0,Y 102.298,Z 444.469,A -85,B 0,C 180,E1 -27953.045,E2 -27953.045} C_VEL
LIN {X 0,Y 101.977,Z 446.175,A -85,B 0,C 180,E1 -27954.137,E2 -27954.137} C_VEL
LIN {X 0,Y 96.212,Z 455.901,A -85,B 0,C 180,E1 -27959.244,E2 -27959.244} C_VEL
LIN {X 0,Y 96.136,Z 456.019,A -85,B 0,C 180,E1 -27959.316,E2 -27959.316} C_VEL
LIN {X 0,Y 93.222,Z 459.745,A -85,B 0,C 180,E1 -27961.471,E2 -27961.471} C_VEL
LIN {X 0,Y 87.129,Z 465.509,A -85,B 0,C 180,E1 -27964.855,E2 -27964.855} C_VEL
LIN {X 0,Y 81.179,Z 470.601,A -85,B 0,C 180,E1 -27968.995,E2 -27968.995} C_VEL
LIN {X 0,Y 78.64,Z 473.272,A -85,B 0,C 180,E1 -27972.304,E2 -27972.304} C_VEL
LIN {X 0,Y 75.645,Z 477.524,A -85,B 0,C 180,E1 -27979.287,E2 -27979.287} C_VEL
LIN {X 0,Y 73.45,Z 481.047,A -85,B 0,C 180,E1 -27987.254,E2 -27987.254} C_VEL
LIN {X 0,Y 72.745,Z 483.554,A -85,B 0,C 180,E1 -27995.54,E2 -27995.54} C_VEL
LIN {X 0,Y 73.014,Z 484.724,A -85,B 0,C 180,E1 -28001.095,E2 -28001.095} C_VEL
LIN {X 0,Y 75.09,Z 485.878,A -85,B 0,C 180,E1 -28011.982,E2 -28011.982} C_VEL
LIN {X 0,Y 77.002,Z 485.885,A -85,B 0,C 180,E1 -28017.148,E2 -28017.148} C_VEL
LIN {X 0,Y 79.416,Z 485.487,A -85,B 0,C 180,E1 -28022.067,E2 -28022.067} C_VEL
LIN {X 0,Y 85.736,Z 483.452,A -85,B 0,C 180,E1 -28030.974,E2 -28030.974} C_VEL
LIN {X 0,Y 89.883,Z 481.667,A -85,B 0,C 180,E1 -28035.272,E2 -28035.272} C_VEL
LIN {X 0,Y 95.838,Z 478.532,A -85,B 0,C 180,E1 -28040.348,E2 -28040.348} C_VEL
LIN {X 0,Y 102.838,Z 474.124,A -85,B 0,C 180,E1 -28045.088,E2 -28045.088} C_VEL
LIN {X 0,Y 107.812,Z 470.476,A -85,B 0,C 180,E1 -28047.929,E2 -28047.929} C_VEL
LIN {X 0,Y 109.526,Z 469.023,A -85,B 0,C 180,E1 -28049.112,E2 -28049.112} C_VEL
LIN {X 0,Y 110.837,Z 466.099,A -85,B 0,C 180,E1 -28053.648,E2 -28053.648} C_VEL
LIN {X 0,Y 111.835,Z 463.533,A -85,B 0,C 180,E1 -28057.848,E2 -28057.848} C_VEL
LIN {X 0,Y 112.475,Z 461.458,A -85,B 0,C 180,E1 -28061.794,E2 -28061.794} C_VEL
LIN {X 0,Y 112.997,Z 459.69,A -85,B 0,C 180,E1 -28065.593,E2 -28065.593} C_VEL
LIN {X 0,Y 113.78,Z 457.593,A -85,B 0,C 180,E1 -28071.208,E2 -28071.208} C_VEL
LIN {X 0,Y 114.766,Z 456.101,A -85,B 0,C 180,E1 -28076.488,E2 -28076.488} C_VEL
LIN {X 0,Y 115.57,Z 455.422,A -85,B 0,C 180,E1 -28079.999,E2 -28079.999} C_VEL
LIN {X 0,Y 115.358,Z 456.234,A -85,B 0,C 180,E1 -28083.492,E2 -28083.492} C_VEL
LIN {X 0,Y 114.92,Z 457.722,A -85,B 0,C 180,E1 -28087.025,E2 -28087.025} C_VEL
LIN {X 0,Y 114.283,Z 460.696,A -85,B 0,C 180,E1 -28092.248,E2 -28092.248} C_VEL
LIN {X 0,Y 113.539,Z 464.885,A -85,B 0,C 180,E1 -28098.028,E2 -28098.028} C_VEL
LIN {X 0,Y 112.823,Z 468.335,A -85,B 0,C 180,E1 -28101.947,E2 -28101.947} C_VEL
LIN {X 0,Y 111.771,Z 472.426,A -85,B 0,C 180,E1 -28106.113,E2 -28106.113} C_VEL
LIN {X 0,Y 109.597,Z 475.512,A -85,B 0,C 180,E1 -28108.154,E2 -28108.154} C_VEL
LIN {X 0,Y 103.579,Z 482.465,A -85,B 0,C 180,E1 -28112.875,E2 -28112.875} C_VEL
LIN {X 0,Y 97.658,Z 488.218,A -85,B 0,C 180,E1 -28117.668,E2 -28117.668} C_VEL
LIN {X 0,Y 93.161,Z 491.684,A -85,B 0,C 180,E1 -28121.033,E2 -28121.033} C_VEL
LIN {X 0,Y 86.522,Z 495.866,A -85,B 0,C 180,E1 -28126.34,E2 -28126.34} C_VEL
LIN {X 0,Y 80.796,Z 499.036,A -85,B 0,C 180,E1 -28132.495,E2 -28132.495} C_VEL
LIN {X 0,Y 74.974,Z 501.803,A -85,B 0,C 180,E1 -28142.055,E2 -28142.055} C_VEL
LIN {X 0,Y 71.799,Z 503.073,A -85,B 0,C 180,E1 -28152.928,E2 -28152.928} C_VEL
LIN {X 0,Y 71.286,Z 503.045,A -85,B 0,C 180,E1 -28160.357,E2 -28160.357} C_VEL
LIN {X 0,Y 71.49,Z 502.771,A -85,B 0,C 180,E1 -28164.362,E2 -28164.362} C_VEL
LIN {X 0,Y 71.892,Z 501.974,A -85,B 0,C 180,E1 -28170.004,E2 -28170.004} C_VEL
LIN {X 0,Y 71.186,Z 499.445,A -85,B 0,C 180,E1 -28179.157,E2 -28179.157} C_VEL
LIN {X 0,Y 71.764,Z 496.295,A -85,B 0,C 180,E1 -28187.09,E2 -28187.09} C_VEL
LIN {X 0,Y 73.807,Z 491.837,A -85,B 0,C 180,E1 -28195.376,E2 -28195.376} C_VEL
LIN {X 0,Y 78.139,Z 485.153,A -85,B 0,C 180,E1 -28204.208,E2 -28204.208} C_VEL
LIN {X 0,Y 80.465,Z 481.686,A -85,B 0,C 180,E1 -28207.695,E2 -28207.695} C_VEL
LIN {X 0,Y 84.905,Z 473.229,A -85,B 0,C 180,E1 -28214.72,E2 -28214.72} C_VEL
LIN {X 0,Y 89.134,Z 464.539,A -85,B 0,C 180,E1 -28220.248,E2 -28220.248} C_VEL
LIN {X 0,Y 93.163,Z 454.957,A -85,B 0,C 180,E1 -28225.128,E2 -28225.128} C_VEL
LIN {X 0,Y 96.21,Z 445.611,A -85,B 0,C 180,E1 -28229.248,E2 -28229.248} C_VEL
LIN {X 0,Y 96.557,Z 444.063,A -85,B 0,C 180,E1 -28229.974,E2 -28229.974} C_VEL
LIN {X 0,Y 95.863,Z 436.378,A -85,B 0,C 180,E1 -28235.273,E2 -28235.273} C_VEL
LIN {X 0,Y 94.996,Z 431.256,A -85,B 0,C 180,E1 -28239.427,E2 -28239.427} C_VEL
LIN {X 0,Y 94.344,Z 427.63,A -85,B 0,C 180,E1 -28242.665,E2 -28242.665} C_VEL
LIN {X 0,Y 93.326,Z 423.844,A -85,B 0,C 180,E1 -28246.944,E2 -28246.944} C_VEL
LIN {X 0,Y 91.365,Z 419.499,A -85,B 0,C 180,E1 -28255.589,E2 -28255.589} C_VEL
LIN {X 0,Y 90.67,Z 418.481,A -85,B 0,C 180,E1 -28260.001,E2 -28260.001} C_VEL
LIN {X 0,Y 89.982,Z 418.567,A -85,B 0,C 180,E1 -28268.988,E2 -28268.988} C_VEL
LIN {X 0,Y 90.258,Z 419.073,A -85,B 0,C 180,E1 -28273.51,E2 -28273.51} C_VEL
LIN {X 0,Y 90.686,Z 420.462,A -85,B 0,C 180,E1 -28278.06,E2 -28278.06} C_VEL
LIN {X 0,Y 91.849,Z 423.43,A -85,B 0,C 180,E1 -28284.889,E2 -28284.889} C_VEL
LIN {X 0,Y 93.309,Z 427.94,A -85,B 0,C 180,E1 -28291.82,E2 -28291.82} C_VEL
LIN {X 0,Y 94.705,Z 432.89,A -85,B 0,C 180,E1 -28297.871,E2 -28297.871} C_VEL
LIN {X 0,Y 95.91,Z 439.051,A -85,B 0,C 180,E1 -28304.116,E2 -28304.116} C_VEL
LIN {X 0,Y 96.301,Z 444.413,A -85,B 0,C 180,E1 -28308.938,E2 -28308.938} C_VEL
LIN {X 0,Y 96.308,Z 447.582,A -85,B 0,C 180,E1 -28311.66,E2 -28311.66} C_VEL
LIN {X 0,Y 90.243,Z 457.205,A -85,B 0,C 180,E1 -28316.961,E2 -28316.961} C_VEL
LIN {X 0,Y 84.753,Z 464.961,A -85,B 0,C 180,E1 -28322.862,E2 -28322.862} C_VEL
LIN {X 0,Y 80.211,Z 471.151,A -85,B 0,C 180,E1 -28329.48,E2 -28329.48} C_VEL
LIN {X 0,Y 78.64,Z 473.272,A -85,B 0,C 180,E1 -28332.304,E2 -28332.304} C_VEL
LIN {X 0,Y 76.267,Z 475.786,A -85,B 0,C 180,E1 -28335.878,E2 -28335.878} C_VEL
LIN {X 0,Y 71.143,Z 479.482,A -85,B 0,C 180,E1 -28341.839,E2 -28341.839} C_VEL
LIN {X 0,Y 66.761,Z 482.546,A -85,B 0,C 180,E1 -28348.809,E2 -28348.809} C_VEL
LIN {X 0,Y 65.71,Z 483.916,A -85,B 0,C 180,E1 -28353.685,E2 -28353.685} C_VEL
LIN {X 0,Y 66.067,Z 485.66,A -85,B 0,C 180,E1 -28362.279,E2 -28362.279} C_VEL
LIN {X 0,Y 68.533,Z 486.771,A -85,B 0,C 180,E1 -28374.213,E2 -28374.213} C_VEL
LIN {X 0,Y 70.727,Z 486.753,A -85,B 0,C 180,E1 -28379.786,E2 -28379.786} C_VEL
LIN {X 0,Y 73.463,Z 486.31,A -85,B 0,C 180,E1 -28385.025,E2 -28385.025} C_VEL
LIN {X 0,Y 80.494,Z 484.224,A -85,B 0,C 180,E1 -28394.301,E2 -28394.301} C_VEL
LIN {X 0,Y 86.81,Z 481.55,A -85,B 0,C 180,E1 -28400.268,E2 -28400.268} C_VEL
LIN {X 0,Y 93.864,Z 477.84,A -85,B 0,C 180,E1 -28405.443,E2 -28405.443} C_VEL
LIN {X 0,Y 101.522,Z 472.978,A -85,B 0,C 180,E1 -28409.915,E2 -28409.915} C_VEL
LIN {X 0,Y 103.907,Z 471.039,A -85,B 0,C 180,E1 -28411.74,E2 -28411.74} C_VEL
LIN {X 0,Y 105.406,Z 468.454,A -85,B 0,C 180,E1 -28416.417,E2 -28416.417} C_VEL
LIN {X 0,Y 106.443,Z 466.319,A -85,B 0,C 180,E1 -28420.722,E2 -28420.722} C_VEL
LIN {X 0,Y 107.192,Z 464.611,A -85,B 0,C 180,E1 -28424.795,E2 -28424.795} C_VEL
LIN {X 0,Y 107.931,Z 463.2,A -85,B 0,C 180,E1 -28428.734,E2 -28428.734} C_VEL
LIN {X 0,Y 108.674,Z 462.02,A -85,B 0,C 180,E1 -28432.568,E2 -28432.568} C_VEL
LIN {X 0,Y 110.455,Z 460.455,A -85,B 0,C 180,E1 -28439.999,E2 -28439.999} C_VEL
LIN {X 0,Y 110.147,Z 461.371,A -85,B 0,C 180,E1 -28443.657,E2 -28443.657} C_VEL
LIN {X 0,Y 109.567,Z 462.969,A -85,B 0,C 180,E1 -28447.37,E2 -28447.37} C_VEL
LIN {X 0,Y 109.021,Z 464.968,A -85,B 0,C 180,E1 -28451.15,E2 -28451.15} C_VEL
LIN {X 0,Y 107.974,Z 468.843,A -85,B 0,C 180,E1 -28457.031,E2 -28457.031} C_VEL
LIN {X 0,Y 106.541,Z 473.374,A -85,B 0,C 180,E1 -28462.563,E2 -28462.563} C_VEL
LIN {X 0,Y 105.759,Z 475.281,A -85,B 0,C 180,E1 -28464.566,E2 -28464.566} C_VEL
LIN {X 0,Y 100.355,Z 481.116,A -85,B 0,C 180,E1 -28468.655,E2 -28468.655} C_VEL
LIN {X 0,Y 93.291,Z 487.55,A -85,B 0,C 180,E1 -28474.043,E2 -28474.043} C_VEL
LIN {X 0,Y 88.607,Z 490.987,A -85,B 0,C 180,E1 -28477.523,E2 -28477.523} C_VEL
LIN {X 0,Y 81.506,Z 495.127,A -85,B 0,C 180,E1 -28482.873,E2 -28482.873} C_VEL
LIN {X 0,Y 75.261,Z 498.263,A -85,B 0,C 180,E1 -28489.186,E2 -28489.186} C_VEL
LIN {X 0,Y 68.738,Z 500.973,A -85,B 0,C 180,E1 -28499.26,E2 -28499.26} C_VEL
LIN {X 0,Y 64.999,Z 502.196,A -85,B 0,C 180,E1 -28511.077,E2 -28511.077} C_VEL
LIN {X 0,Y 64.418,Z 501.837,A -85,B 0,C 180,E1 -28523.741,E2 -28523.741} C_VEL
LIN {X 0,Y 64.785,Z 501.02,A -85,B 0,C 180,E1 -28530.005,E2 -28530.005} C_VEL
LIN {X 0,Y 64.119,Z 498.657,A -85,B 0,C 180,E1 -28539.439,E2 -28539.439} C_VEL
LIN {X 0,Y 64.927,Z 495.238,A -85,B 0,C 180,E1 -28548.954,E2 -28548.954} C_VEL
LIN {X 0,Y 67.38,Z 490.729,A -85,B 0,C 180,E1 -28557.998,E2 -28557.998} C_VEL
LIN {X 0,Y 71.483,Z 485.031,A -85,B 0,C 180,E1 -28566.155,E2 -28566.155} C_VEL
LIN {X 0,Y 74.011,Z 481.67,A -85,B 0,C 180,E1 -28569.87,E2 -28569.87} C_VEL
LIN {X 0,Y 78.865,Z 473.462,A -85,B 0,C 180,E1 -28577.329,E2 -28577.329} C_VEL
LIN {X 0,Y 83.286,Z 465.413,A -85,B 0,C 180,E1 -28582.85,E2 -28582.85} C_VEL
LIN {X 0,Y 87.93,Z 455.677,A -85,B 0,C 180,E1 -28588.134,E2 -28588.134} C_VEL
LIN {X 0,Y 90.81,Z 448.274,A -85,B 0,C 180,E1 -28591.651,E2 -28591.651} C_VEL
LIN {X 0,Y 91.216,Z 446.674,A -85,B 0,C 180,E1 -28592.466,E2 -28592.466} C_VEL
LIN {X 0,Y 90.963,Z 439.559,A -85,B 0,C 180,E1 -28598.002,E2 -28598.002} C_VEL
LIN {X 0,Y 90.29,Z 432.896,A -85,B 0,C 180,E1 -28604.192,E2 -28604.192} C_VEL
LIN {X 0,Y 89.538,Z 429.38,A -85,B 0,C 180,E1 -28608.684,E2 -28608.684} C_VEL
LIN {X 0,Y 88.324,Z 426.116,A -85,B 0,C 180,E1 -28615.437,E2 -28615.437} C_VEL
LIN {X 0,Y 87.694,Z 424.97,A -85,B 0,C 180,E1 -28620.001,E2 -28620.001} C_VEL
LIN {X 0,Y 86.959,Z 425.022,A -85,B 0,C 180,E1 -28629.303,E2 -28629.303} C_VEL
LIN {X 0,Y 87.152,Z 425.833,A -85,B 0,C 180,E1 -28634.592,E2 -28634.592} C_VEL
LIN {X 0,Y 87.981,Z 429.084,A -85,B 0,C 180,E1 -28643.542,E2 -28643.542} C_VEL
LIN {X 0,Y 88.992,Z 433.383,A -85,B 0,C 180,E1 -28650.884,E2 -28650.884} C_VEL
LIN {X 0,Y 89.806,Z 437.503,A -85,B 0,C 180,E1 -28656.419,E2 -28656.419} C_VEL
LIN {X 0,Y 90.38,Z 441.804,A -85,B 0,C 180,E1 -28661.372,E2 -28661.372} C_VEL
LIN {X 0,Y 90.589,Z 446.965,A -85,B 0,C 180,E1 -28666.642,E2 -28666.642} C_VEL
LIN {X 0,Y 90.521,Z 449.163,A -85,B 0,C 180,E1 -28668.791,E2 -28668.791} C_VEL
LIN {X 0,Y 89.796,Z 450.769,A -85,B 0,C 180,E1 -28669.823,E2 -28669.823} C_VEL
LIN {X 0,Y 84.436,Z 458.51,A -85,B 0,C 180,E1 -28674.359,E2 -28674.359} C_VEL
LIN {X 0,Y 78.566,Z 466.156,A -85,B 0,C 180,E1 -28680.524,E2 -28680.524} C_VEL
LIN {X 0,Y 73.644,Z 472.288,A -85,B 0,C 180,E1 -28687.555,E2 -28687.555} C_VEL
LIN {X 0,Y 69.733,Z 477.187,A -85,B 0,C 180,E1 -28695.402,E2 -28695.402} C_VEL
LIN {X 0,Y 67.018,Z 480.997,A -85,B 0,C 180,E1 -28703.976,E2 -28703.976} C_VEL
LIN {X 0,Y 65.71,Z 483.916,A -85,B 0,C 180,E1 -28713.685,E2 -28713.685} C_VEL
LIN {X 0,Y 65.101,Z 485.133,A -85,B 0,C 180,E1 -28718.723,E2 -28718.723} C_VEL
LIN {X 0,Y 63.203,Z 486.687,A -85,B 0,C 180,E1 -28727.321,E2 -28727.321} C_VEL
LIN {X 0,Y 62.49,Z 487.451,A -85,B 0,C 180,E1 -28734.55,E2 -28734.55} C_VEL
LIN {X 0,Y 63.347,Z 487.659,A -85,B 0,C 180,E1 -28739.907,E2 -28739.907} C_VEL
LIN {X 0,Y 64.002,Z 487.622,A -85,B 0,C 180,E1 -28741.59,E2 -28741.59} C_VEL
LIN {X 0,Y 67.748,Z 487.132,A -85,B 0,C 180,E1 -28748.488,E2 -28748.488} C_VEL
LIN {X 0,Y 71.383,Z 486.268,A -85,B 0,C 180,E1 -28753.56,E2 -28753.56} C_VEL
LIN {X 0,Y 79.647,Z 483.474,A -85,B 0,C 180,E1 -28761.852,E2 -28761.852} C_VEL
LIN {X 0,Y 87.405,Z 479.9,A -85,B 0,C 180,E1 -28767.588,E2 -28767.588} C_VEL
LIN {X 0,Y 95.381,Z 475.37,A -85,B 0,C 180,E1 -28772.147,E2 -28772.147} C_VEL
LIN {X 0,Y 97.895,Z 473.7,A -85,B 0,C 180,E1 -28773.613,E2 -28773.613} C_VEL
LIN {X 0,Y 99.245,Z 471.999,A -85,B 0,C 180,E1 -28777.005,E2 -28777.005} C_VEL
LIN {X 0,Y 100.033,Z 470.902,A -85,B 0,C 180,E1 -28779.433,E2 -28779.433} C_VEL
LIN {X 0,Y 101.517,Z 468.548,A -85,B 0,C 180,E1 -28785.734,E2 -28785.734} C_VEL
LIN {X 0,Y 102.952,Z 466.71,A -85,B 0,C 180,E1 -28792.152,E2 -28792.152} C_VEL
LIN {X 0,Y 103.94,Z 465.861,A -85,B 0,C 180,E1 -28796.122,E2 -28796.122} C_VEL
LIN {X 0,Y 105.057,Z 465.22,A -85,B 0,C 180,E1 -28799.999,E2 -28799.999} C_VEL
LIN {X 0,Y 104.634,Z 466.242,A -85,B 0,C 180,E1 -28803.85,E2 -28803.85} C_VEL
LIN {X 0,Y 103.582,Z 468.85,A -85,B 0,C 180,E1 -28809.765,E2 -28809.765} C_VEL
LIN {X 0,Y 102.235,Z 472.542,A -85,B 0,C 180,E1 -28815.96,E2 -28815.96} C_VEL
LIN {X 0,Y 100.464,Z 476.721,A -85,B 0,C 180,E1 -28821.605,E2 -28821.605} C_VEL
LIN {X 0,Y 99.274,Z 478.256,A -85,B 0,C 180,E1 -28823.034,E2 -28823.034} C_VEL
LIN {X 0,Y 91.702,Z 484.996,A -85,B 0,C 180,E1 -28828.341,E2 -28828.341} C_VEL
LIN {X 0,Y 86.882,Z 488.643,A -85,B 0,C 180,E1 -28831.865,E2 -28831.865} C_VEL
LIN {X 0,Y 81.824,Z 491.791,A -85,B 0,C 180,E1 -28835.323,E2 -28835.323} C_VEL
LIN {X 0,Y 72.658,Z 496.325,A -85,B 0,C 180,E1 -28842.615,E2 -28842.615} C_VEL
LIN {X 0,Y 66.09,Z 499.005,A -85,B 0,C 180,E1 -28850.36,E2 -28850.36} C_VEL
LIN {X 0,Y 60.095,Z 500.919,A -85,B 0,C 180,E1 -28862.114,E2 -28862.114} C_VEL
LIN {X 0,Y 58.295,Z 501.311,A -85,B 0,C 180,E1 -28868.802,E2 -28868.802} C_VEL
LIN {X 0,Y 57.355,Z 500.904,A -85,B 0,C 180,E1 -28882.967,E2 -28882.967} C_VEL
LIN {X 0,Y 57.679,Z 500.065,A -85,B 0,C 180,E1 -28890.005,E2 -28890.005} C_VEL
LIN {X 0,Y 57.053,Z 497.871,A -85,B 0,C 180,E1 -28899.784,E2 -28899.784} C_VEL
LIN {X 0,Y 58.162,Z 494.178,A -85,B 0,C 180,E1 -28911.259,E2 -28911.259} C_VEL
LIN {X 0,Y 61.139,Z 489.624,A -85,B 0,C 180,E1 -28921.156,E2 -28921.156} C_VEL
LIN {X 0,Y 65.849,Z 483.876,A -85,B 0,C 180,E1 -28929.825,E2 -28929.825} C_VEL
LIN {X 0,Y 68.822,Z 479.963,A -85,B 0,C 180,E1 -28934.373,E2 -28934.373} C_VEL
LIN {X 0,Y 73.998,Z 472.116,A -85,B 0,C 180,E1 -28941.592,E2 -28941.592} C_VEL
LIN {X 0,Y 78.51,Z 464.71,A -85,B 0,C 180,E1 -28946.799,E2 -28946.799} C_VEL
LIN {X 0,Y 83.483,Z 455.224,A -85,B 0,C 180,E1 -28952.128,E2 -28952.128} C_VEL
LIN {X 0,Y 85.643,Z 450.396,A -85,B 0,C 180,E1 -28954.52,E2 -28954.52} C_VEL
LIN {X 0,Y 86.046,Z 447.546,A -85,B 0,C 180,E1 -28956.673,E2 -28956.673} C_VEL
LIN {X 0,Y 86.136,Z 442.743,A -85,B 0,C 180,E1 -28960.953,E2 -28960.953} C_VEL
LIN {X 0,Y 86.025,Z 438.01,A -85,B 0,C 180,E1 -28965.814,E2 -28965.814} C_VEL
LIN {X 0,Y 85.553,Z 434.723,A -85,B 0,C 180,E1 -28970.545,E2 -28970.545} C_VEL
LIN {X 0,Y 84.908,Z 432.576,A -85,B 0,C 180,E1 -28975.253,E2 -28975.253} C_VEL
LIN {X 0,Y 84.342,Z 431.238,A -85,B 0,C 180,E1 -28980.242,E2 -28980.242} C_VEL
LIN {X 0,Y 83.579,Z 431.321,A -85,B 0,C 180,E1 -28989.683,E2 -28989.683} C_VEL
LIN {X 0,Y 83.59,Z 432.089,A -85,B 0,C 180,E1 -28994.611,E2 -28994.611} C_VEL
LIN {X 0,Y 83.96,Z 434.969,A -85,B 0,C 180,E1 -29002.952,E2 -29002.952} C_VEL
LIN {X 0,Y 84.487,Z 438.692,A -85,B 0,C 180,E1 -29009.942,E2 -29009.942} C_VEL
LIN {X 0,Y 84.861,Z 442.427,A -85,B 0,C 180,E1 -29015.432,E2 -29015.432} C_VEL
LIN {X 0,Y 85.053,Z 447.146,A -85,B 0,C 180,E1 -29021.381,E2 -29021.381} C_VEL
LIN {X 0,Y 84.816,Z 451.047,A -85,B 0,C 180,E1 -29025.724,E2 -29025.724} C_VEL
LIN {X 0,Y 84.409,Z 452.363,A -85,B 0,C 180,E1 -29026.857,E2 -29026.857} C_VEL
LIN {X 0,Y 77.69,Z 461.162,A -85,B 0,C 180,E1 -29032.361,E2 -29032.361} C_VEL
LIN {X 0,Y 71.535,Z 468.464,A -85,B 0,C 180,E1 -29038.945,E2 -29038.945} C_VEL
LIN {X 0,Y 65.657,Z 475.183,A -85,B 0,C 180,E1 -29047.993,E2 -29047.993} C_VEL
LIN {X 0,Y 61.79,Z 479.653,A -85,B 0,C 180,E1 -29056.846,E2 -29056.846} C_VEL
LIN {X 0,Y 59.996,Z 482.027,A -85,B 0,C 180,E1 -29063.268,E2 -29063.268} C_VEL
LIN {X 0,Y 58.67,Z 484.732,A -85,B 0,C 180,E1 -29073.362,E2 -29073.362} C_VEL
LIN {X 0,Y 59.155,Z 486.595,A -85,B 0,C 180,E1 -29083.741,E2 -29083.741} C_VEL
LIN {X 0,Y 62.109,Z 487.662,A -85,B 0,C 180,E1 -29096.907,E2 -29096.907} C_VEL
LIN {X 0,Y 64.002,Z 487.622,A -85,B 0,C 180,E1 -29101.59,E2 -29101.59} C_VEL
LIN {X 0,Y 65.875,Z 487.526,A -85,B 0,C 180,E1 -29106.53,E2 -29106.53} C_VEL
LIN {X 0,Y 68.319,Z 486.994,A -85,B 0,C 180,E1 -29114.723,E2 -29114.723} C_VEL
LIN {X 0,Y 70.953,Z 486.013,A -85,B 0,C 180,E1 -29120.848,E2 -29120.848} C_VEL
LIN {X 0,Y 73.933,Z 484.818,A -85,B 0,C 180,E1 -29124.786,E2 -29124.786} C_VEL
LIN {X 0,Y 75.17,Z 484.316,A -85,B 0,C 180,E1 -29125.903,E2 -29125.903} C_VEL
LIN {X 0,Y 83.795,Z 480.578,A -85,B 0,C 180,E1 -29131.713,E2 -29131.713} C_VEL
LIN {X 0,Y 92.213,Z 476.002,A -85,B 0,C 180,E1 -29136.137,E2 -29136.137} C_VEL
LIN {X 0,Y 93.006,Z 475.259,A -85,B 0,C 180,E1 -29137.8,E2 -29137.8} C_VEL
LIN {X 0,Y 94.96,Z 473.067,A -85,B 0,C 180,E1 -29144.171,E2 -29144.171} C_VEL
LIN {X 0,Y 95.844,Z 472.111,A -85,B 0,C 180,E1 -29147.291,E2 -29147.291} C_VEL
LIN {X 0,Y 96.936,Z 471.102,A -85,B 0,C 180,E1 -29151.662,E2 -29151.662} C_VEL
LIN {X 0,Y 98.499,Z 470.05,A -85,B 0,C 180,E1 -29157.262,E2 -29157.262} C_VEL
LIN {X 0,Y 99.369,Z 469.7,A -85,B 0,C 180,E1 -29159.999,E2 -29159.999} C_VEL
LIN {X 0,Y 98.703,Z 470.995,A -85,B 0,C 180,E1 -29164.589,E2 -29164.589} C_VEL
LIN {X 0,Y 97.983,Z 472.464,A -85,B 0,C 180,E1 -29168.247,E2 -29168.247} C_VEL
LIN {X 0,Y 96.909,Z 474.682,A -85,B 0,C 180,E1 -29172.565,E2 -29172.565} C_VEL
LIN {X 0,Y 95.55,Z 477.419,A -85,B 0,C 180,E1 -29177.109,E2 -29177.109} C_VEL
LIN {X 0,Y 94.98,Z 478.479,A -85,B 0,C 180,E1 -29178.704,E2 -29178.704} C_VEL
LIN {X 0,Y 93.77,Z 480.023,A -85,B 0,C 180,E1 -29180.478,E2 -29180.478} C_VEL
LIN {X 0,Y 85.817,Z 486.208,A -85,B 0,C 180,E1 -29185.738,E2 -29185.738} C_VEL
LIN {X 0,Y 80.582,Z 489.585,A -85,B 0,C 180,E1 -29189.297,E2 -29189.297} C_VEL
LIN {X 0,Y 72.541,Z 493.648,A -85,B 0,C 180,E1 -29194.57,E2 -29194.57} C_VEL
LIN {X 0,Y 65.124,Z 496.694,A -85,B 0,C 180,E1 -29200.944,E2 -29200.944} C_VEL
LIN {X 0,Y 56.925,Z 499.313,A -85,B 0,C 180,E1 -29211.887,E2 -29211.887} C_VEL
LIN {X 0,Y 53.884,Z 500.068,A -85,B 0,C 180,E1 -29218.559,E2 -29218.559} C_VEL
LIN {X 0,Y 50.468,Z 500.376,A -85,B 0,C 180,E1 -29233.834,E2 -29233.834} C_VEL
LIN {X 0,Y 50.272,Z 499.967,A -85,B 0,C 180,E1 -29241.97,E2 -29241.97} C_VEL
LIN {X 0,Y 50.552,Z 499.109,A -85,B 0,C 180,E1 -29250.006,E2 -29250.006} C_VEL
LIN {X 0,Y 49.988,Z 497.087,A -85,B 0,C 180,E1 -29260.219,E2 -29260.219} C_VEL
LIN {X 0,Y 51.54,Z 493.122,A -85,B 0,C 180,E1 -29274.153,E2 -29274.153} C_VEL
LIN {X 0,Y 55.136,Z 488.52,A -85,B 0,C 180,E1 -29285.008,E2 -29285.008} C_VEL
LIN {X 0,Y 60.512,Z 482.716,A -85,B 0,C 180,E1 -29294.182,E2 -29294.182} C_VEL
LIN {X 0,Y 65.3,Z 476.584,A -85,B 0,C 180,E1 -29301.294,E2 -29301.294} C_VEL
LIN {X 0,Y 70.715,Z 469.181,A -85,B 0,C 180,E1 -29307.655,E2 -29307.655} C_VEL
LIN {X 0,Y 76.859,Z 459.527,A -85,B 0,C 180,E1 -29313.932,E2 -29313.932} C_VEL
LIN {X 0,Y 80.547,Z 452.664,A -85,B 0,C 180,E1 -29317.625,E2 -29317.625} C_VEL
LIN {X 0,Y 81.118,Z 449.024,A -85,B 0,C 180,E1 -29320.928,E2 -29320.928} C_VEL
LIN {X 0,Y 81.493,Z 444.05,A -85,B 0,C 180,E1 -29326.282,E2 -29326.282} C_VEL
LIN {X 0,Y 81.519,Z 441.216,A -85,B 0,C 180,E1 -29330.072,E2 -29330.072} C_VEL
LIN {X 0,Y 81.126,Z 438.849,A -85,B 0,C 180,E1 -29335.031,E2 -29335.031} C_VEL
LIN {X 0,Y 80.687,Z 437.414,A -85,B 0,C 180,E1 -29340.001,E2 -29340.001} C_VEL
LIN {X 0,Y 79.888,Z 437.316,A -85,B 0,C 180,E1 -29347.002,E2 -29347.002} C_VEL
LIN {X 0,Y 79.781,Z 437.457,A -85,B 0,C 180,E1 -29350.149,E2 -29350.149} C_VEL
LIN {X 0,Y 79.638,Z 438.384,A -85,B 0,C 180,E1 -29355.353,E2 -29355.353} C_VEL
LIN {X 0,Y 79.667,Z 440.755,A -85,B 0,C 180,E1 -29362.562,E2 -29362.562} C_VEL
LIN {X 0,Y 79.773,Z 443.464,A -85,B 0,C 180,E1 -29368.229,E2 -29368.229} C_VEL
LIN {X 0,Y 79.781,Z 447.048,A -85,B 0,C 180,E1 -29374.166,E2 -29374.166} C_VEL
LIN {X 0,Y 79.662,Z 449.84,A -85,B 0,C 180,E1 -29378.14,E2 -29378.14} C_VEL
LIN {X 0,Y 79.176,Z 453.946,A -85,B 0,C 180,E1 -29383.451,E2 -29383.451} C_VEL
LIN {X 0,Y 72.262,Z 462.415,A -85,B 0,C 180,E1 -29388.962,E2 -29388.962} C_VEL
